  MoveL 2095 to (-402.87, 337.02, -18.74) mm, rotated rx -180 ry 0 rz 0.01 deg; joints [35.505, -31.649, 74.768, -134.161, 54.079, 149.801]
  MoveL 2096 to (-403.75, 334.43, -18.84) mm, rotated rx -180 ry 0 rz 0.01 deg; joints [35.421, -31.691, 74.866, -134.279, 54.073, 149.904]
  MoveL 2097 to (-403.78, 333.95, -18.85) mm, rotated rx -180 ry 0 rz 0.01 deg; joints [35.407, -31.706, 74.899, -134.302, 54.079, 149.928]
  MoveL 2098 to (-403.79, 333.65, -18.86) mm, rotated rx -180 ry 0 rz 0.01 deg; joints [35.399, -31.715, 74.92, -134.317, 54.083, 149.943]
  MoveL 2099 to (-403.79, 333.05, -18.88) mm, rotated rx -180 ry 0 rz 0.01 deg; joints [35.384, -31.736, 74.964, -134.346, 54.091, 149.974]
  MoveL 2100 to (-401.25, 328.08, -19.09) mm, rotated rx 180 ry 0 rz 0.01 deg; joints [35.3, -32.028, 75.587, -134.605, 54.28, 150.319]
  MoveL 2101 to (-395.74, 327.2, -19.29) mm, rotated rx -180 ry 0 rz 0.01 deg; joints [35.38, -32.323, 76.213, -134.688, 54.554, 150.557]
  MoveL 2102 to (-391.79, 331.15, -19.49) mm, rotated rx 180 ry 0 rz 0.01 deg; joints [35.56, -32.373, 76.328, -134.532, 54.691, 150.502]
  MoveL 2103 to (-392.66, 336.66, -19.69) mm, rotated rx -180 ry 0 rz 0.01 deg; joints [35.689, -32.13, 75.838, -134.27, 54.584, 150.205]
  MoveL 2104 to (-397.64, 339.2, -19.9) mm, rotated rx 180 ry 0 rz 0.01 deg; joints [35.662, -31.785, 75.142, -134.119, 54.326, 149.913]
  MoveL 2105 to (-398.51, 339.2, -19.93) mm, rotated rx -180 ry 0 rz 0.01 deg; joints [35.645, -31.741, 75.052, -134.113, 54.286, 149.884]
  MoveL 2106 to (-399.34, 339.13, -19.95) mm, rotated rx 180 ry 0 rz 0.01 deg; joints [35.628, -31.7, 74.972, -134.111, 54.249, 149.859]
  MoveL 2107 to (-399.69, 339.08, -19.97) mm, rotated rx 180 ry 0 rz 0.01 deg; joints [35.62, -31.684, 74.939, -134.111, 54.233, 149.85]
  MoveL 2108 to (-400.55, 338.85, -20) mm, rotated rx 180 ry 0 rz 0.01 deg; joints [35.598, -31.647, 74.867, -134.116, 54.197, 149.832]
  MoveL 2109 to (-400.6, 338.83, -20) mm, rotated rx 180 ry 0 rz 0.01 deg; joints [35.596, -31.646, 74.864, -134.116, 54.195, 149.832]
  MoveL 2110 to (-400.13, 339.01, -20) mm, rotated rx 180 ry 0 rz 0.01 deg; joints [35.61, -31.663, 74.899, -134.112, 54.215, 149.839]
  MoveL 2111 to (-398.92, 339.2, -20) mm, rotated rx 180 ry 0 rz 0.01 deg; joints [35.637, -31.717, 75.009, -134.112, 54.269, 149.872]
  MoveL 2112 to (-213.2, 339.2, -20) mm, rotated rx 180 ry 0 rz 0.01 deg; joints [39.463, -39.848, 91.814, -134.031, 62.159, 155.085]
  MoveL 2113 to (-213.59, 339.14, -20) mm, rotated rx 180 ry 0 rz 0.01 deg; joints [39.452, -39.834, 91.787, -134.036, 62.144, 155.079]
  MoveL 2114 to (-214.1, 339.03, -20) mm, rotated rx 180 ry 0 rz 0.01 deg; joints [39.438, -39.818, 91.754, -134.044, 62.126, 155.072]
  MoveL 2115 to (-215.18, 338.68, -20) mm, rotated rx 180 ry 0 rz 0.01 deg; joints [39.404, -39.787, 91.689, -134.066, 62.088, 155.061]
  MoveL 2116 to (-215.68, 338.49, -20) mm, rotated rx -180 ry 0 rz 0.01 deg; joints [39.388, -39.774, 91.662, -134.077, 62.071, 155.058]
  MoveL 2117 to (-226.92, 332.89, -20) mm, rotated rx 180 ry 0 rz 0.01 deg; joints [38.984, -39.51, 91.121, -134.381, 61.699, 155.03]
  MoveL 2118 to (-227.59, 332.45, -20) mm, rotated rx -180 ry 0 rz 0.01 deg; joints [38.958, -39.497, 91.095, -134.403, 61.678, 155.033]
  MoveL 2119 to (-228.68, 331.54, -20) mm, rotated rx 180 ry 0 rz 0.01 deg; joints [38.909, -39.483, 91.066, -134.448, 61.646, 155.045]
  MoveL 2120 to (-228.85, 331.38, -20) mm, rotated rx 180 ry 0 rz 0.01 deg; joints [38.901, -39.481, 91.062, -134.455, 61.641, 155.048]
  MoveL 2121 to (-237.26, 323.26, -20) mm, rotated rx -180 ry 0 rz 0.01 deg; joints [38.493, -39.4, 90.906, -134.842, 61.408, 155.189]
  MoveL 2122 to (-237.74, 322.68, -20) mm, rotated rx -180 ry 0 rz 0.01 deg; joints [38.467, -39.399, 90.905, -134.869, 61.396, 155.202]
  MoveL 2123 to (-238.69, 321.23, -20) mm, rotated rx -180 ry 0 rz 0.01 deg; joints [38.406, -39.406, 90.921, -134.934, 61.376, 155.24]
  MoveL 2124 to (-238.83, 321, -20) mm, rotated rx -180 ry 0 rz 0.01 deg; joints [38.397, -39.407, 90.925, -134.945, 61.373, 155.247]
  MoveL 2125 to (-243.98, 311.57, -20) mm, rotated rx 180 ry 0 rz 0.01 deg; joints [38.024, -39.491, 91.112, -135.366, 61.284, 155.517]
  MoveL 2126 to (-244.14, 311.23, -20) mm, rotated rx -180 ry 0 rz 0.01 deg; joints [38.011, -39.495, 91.121, -135.381, 61.281, 155.527]
  MoveL 2127 to (-244.73, 309.78, -20) mm, rotated rx 180 ry 0 rz 0.01 deg; joints [37.958, -39.515, 91.165, -135.445, 61.275, 155.573]
  MoveL 2128 to (-244.95, 309.01, -20) mm, rotated rx 180 ry 0 rz 0.01 deg; joints [37.932, -39.53, 91.197, -135.478, 61.276, 155.6]
  MoveL 2129 to (-246.39, 299.58, -20) mm, rotated rx 180 ry 0 rz 0.01 deg; joints [37.638, -39.756, 91.681, -135.879, 61.334, 155.954]
  MoveL 2130 to (-246.42, 299.36, -20) mm, rotated rx 180 ry 0 rz 0.01 deg; joints [37.631, -39.761, 91.692, -135.888, 61.335, 155.962]
  MoveL 2131 to (-246.51, 298.27, -20) mm, rotated rx -180 ry 0 rz 0.01 deg; joints [37.599, -39.79, 91.754, -135.934, 61.345, 156.004]
  MoveC 2132 to (-246.51, 297.75, -20) mm, rotated rx -180 ry 0 rz 0.01 deg; joints [37.584, -39.805, 91.786, -135.956, 61.351, 156.025] to (-246.44, 297.23, -20) mm, rotated rx -180 ry 0 rz 0.01 deg; joints [37.572, -39.824, 91.825, -135.977, 61.36, 156.048]
  MoveL 2133 to (-245.04, 291.02, -20) mm, rotated rx 180 ry 0 rz 0.01 deg; joints [37.427, -40.063, 92.332, -136.227, 61.492, 156.332]
  MoveL 2134 to (-245.03, 290.96, -20) mm, rotated rx 180 ry 0 rz 0.01 deg; joints [37.426, -40.065, 92.337, -136.229, 61.493, 156.335]
  MoveL 2135 to (-244.07, 287.02, -20) mm, rotated rx 180 ry 0 rz 0.01 deg; joints [37.336, -40.219, 92.663, -136.387, 61.579, 156.515]
  MoveL 2136 to (-243.75, 286.2, -20) mm, rotated rx -180 ry 0 rz 0.01 deg; joints [37.319, -40.255, 92.74, -136.418, 61.602, 156.555]
  MoveL 2137 to (-242.37, 283.67, -20) mm, rotated rx 180 ry 0 rz 0.01 deg; joints [37.277, -40.384, 93.011, -136.515, 61.688, 156.688]
  MoveL 2138 to (-242.16, 283.33, -20) mm, rotated rx -180 ry 0 rz 0.01 deg; joints [37.272, -40.402, 93.049, -136.527, 61.7, 156.706]
  MoveL 2139 to (-239.17, 279.09, -20) mm, rotated rx -180 ry 0 rz 0.01 deg; joints [37.217, -40.642, 93.556, -136.683, 61.871, 156.942]
  MoveL 2140 to (-239, 278.88, -20) mm, rotated rx -180 ry 0 rz 0.01 deg; joints [37.214, -40.655, 93.583, -136.691, 61.88, 156.954]
  MoveL 2141 to (-237.09, 276.58, -20) mm, rotated rx -180 ry 0 rz 0.01 deg; joints [37.19, -40.796, 93.879, -136.773, 61.983, 157.087]
  MoveL 2142 to (-236.75, 276.23, -20) mm, rotated rx -180 ry 0 rz 0.01 deg; joints [37.187, -40.819, 93.928, -136.785, 62.001, 157.108]
  MoveL 2143 to (-236.39, 275.91, -20) mm, rotated rx -180 ry 0 rz 0.01 deg; joints [37.186, -40.842, 93.978, -136.796, 62.02, 157.129]
  MoveL 2144 to (-236.08, 275.67, -20) mm, rotated rx 180 ry 0 rz 0.01 deg; joints [37.186, -40.861, 94.018, -136.804, 62.034, 157.146]
  MoveL 2145 to (-232.45, 273.09, -20) mm, rotated rx -180 ry 0 rz 0.01 deg; joints [37.191, -41.076, 94.469, -136.884, 62.209, 157.326]
  MoveL 2146 to (-232.33, 273.01, -20) mm, rotated rx -180 ry 0 rz 0.01 deg; joints [37.191, -41.083, 94.484, -136.886, 62.215, 157.332]
  MoveL 2147 to (-229.06, 270.9, -20) mm, rotated rx -180 ry 0 rz 0.01 deg; joints [37.202, -41.269, 94.876, -136.949, 62.37, 157.486]
  MoveL 2148 to (-228.75, 270.72, -20) mm, rotated rx 180 ry 0 rz 0.01 deg; joints [37.203, -41.287, 94.912, -136.954, 62.384, 157.499]
  MoveL 2149 to (-227.17, 269.93, -20) mm, rotated rx -180 ry 0 rz 0.01 deg; joints [37.215, -41.37, 95.087, -136.975, 62.456, 157.564]
  MoveL 2150 to (-226.77, 269.76, -20) mm, rotated rx -180 ry 0 rz 0.01 deg; joints [37.219, -41.39, 95.129, -136.979, 62.474, 157.579]
  MoveL 2151 to (-224.72, 269.04, -20) mm, rotated rx 180 ry 0 rz 0.01 deg; joints [37.243, -41.489, 95.337, -136.993, 62.563, 157.651]
  MoveL 2152 to (-224.25, 268.91, -20) mm, rotated rx 180 ry 0 rz 0.01 deg; joints [37.25, -41.511, 95.383, -136.994, 62.583, 157.667]
  MoveL 2153 to (-219.17, 267.91, -20) mm, rotated rx -180 ry 0 rz 0.01 deg; joints [37.332, -41.733, 95.848, -136.995, 62.794, 157.813]
  MoveL 2154 to (-218.97, 267.88, -20) mm, rotated rx 180 ry 0 rz 0.01 deg; joints [37.336, -41.742, 95.866, -136.994, 62.802, 157.819]
  MoveL 2155 to (-215.35, 267.39, -20) mm, rotated rx 180 ry 0 rz 0.01 deg; joints [37.401, -41.893, 96.184, -136.985, 62.95, 157.914]
  MoveL 2156 to (-214.9, 267.36, -20) mm, rotated rx 180 ry 0 rz 0.01 deg; joints [37.41, -41.911, 96.221, -136.982, 62.967, 157.925]
  MoveL 2157 to (-178.62, 267.36, -20) mm, rotated rx 180 ry 0 rz 0.01 deg; joints [38.225, -43.259, 99.04, -136.644, 64.36, 158.668]
  MoveL 2158 to (-178.17, 267.39, -20) mm, rotated rx 180 ry 0 rz 0.01 deg; joints [38.236, -43.275, 99.073, -136.639, 64.376, 158.676]
  MoveL 2159 to (-174.54, 267.88, -20) mm, rotated rx 180 ry 0 rz 0.01 deg; joints [38.334, -43.393, 99.32, -136.581, 64.507, 158.73]
  MoveL 2160 to (-174.34, 267.91, -20) mm, rotated rx -180 ry 0 rz 0.01 deg; joints [38.339, -43.399, 99.333, -136.578, 64.515, 158.733]
  MoveL 2161 to (-169.26, 268.91, -20) mm, rotated rx 180 ry 0 rz 0.01 deg; joints [38.485, -43.555, 99.658, -136.484, 64.694, 158.797]
  MoveL 2162 to (-168.86, 269.01, -20) mm, rotated rx 180 ry 0 rz 0.01 deg; joints [38.497, -43.567, 99.683, -136.476, 64.707, 158.801]
  MoveL 2163 to (-167.47, 269.46, -20) mm, rotated rx -180 ry 0 rz 0.01 deg; joints [38.542, -43.604, 99.76, -136.443, 64.754, 158.811]
  MoveL 2164 to (-167.13, 269.6, -20) mm, rotated rx -180 ry 0 rz 0.01 deg; joints [38.554, -43.613, 99.778, -136.434, 64.765, 158.813]
  MoveL 2165 to (-165.28, 270.43, -20) mm, rotated rx -180 ry 0 rz 0.01 deg; joints [38.621, -43.656, 99.867, -136.38, 64.824, 158.818]
  MoveL 2166 to (-164.86, 270.66, -20) mm, rotated rx -180 ry 0 rz 0.01 deg; joints [38.638, -43.665, 99.885, -136.366, 64.837, 158.818]
  MoveL 2167 to (-161.56, 272.76, -20) mm, rotated rx -180 ry 0 rz 0.01 deg; joints [38.775, -43.724, 100.007, -136.246, 64.935, 158.804]
  MoveL 2168 to (-161.46, 272.83, -20) mm, rotated rx -180 ry 0 rz 0.01 deg; joints [38.78, -43.726, 100.01, -136.242, 64.938, 158.803]
  MoveL 2169 to (-158.56, 274.83, -20) mm, rotated rx 180 ry 0 rz 0.01 deg; joints [38.905, -43.774, 100.107, -136.13, 65.022, 158.786]
  MoveL 2170 to (-158.4, 274.95, -20) mm, rotated rx -180 ry 0 rz 0.01 deg; joints [38.913, -43.776, 100.112, -136.124, 65.026, 158.784]
  MoveL 2171 to (-156.94, 276.09, -20) mm, rotated rx -180 ry 0 rz 0.01 deg; joints [38.98, -43.796, 100.153, -136.062, 65.067, 158.77]
  MoveL 2172 to (-156.45, 276.55, -20) mm, rotated rx -180 ry 0 rz 0.01 deg; joints [39.005, -43.801, 100.161, -136.038, 65.079, 158.762]
  MoveL 2173 to (-155.01, 278.23, -20) mm, rotated rx 180 ry 0 rz 0.01 deg; joints [39.087, -43.805, 100.167, -135.954, 65.112, 158.728]
  MoveL 2174 to (-154.82, 278.47, -20) mm, rotated rx 180 ry 0 rz 0.01 deg; joints [39.098, -43.805, 100.166, -135.943, 65.116, 158.722]
  MoveL 2175 to (-151.36, 283.31, -20) mm, rotated rx 180 ry 0 rz 0.01 deg; joints [39.32, -43.791, 100.13, -135.711, 65.185, 158.608]
  MoveL 2176 to (-151.14, 283.67, -20) mm, rotated rx 180 ry 0 rz 0.01 deg; joints [39.335, -43.789, 100.125, -135.694, 65.189, 158.599]
  MoveL 2177 to (-149.76, 286.2, -20) mm, rotated rx 180 ry 0 rz 0.01 deg; joints [39.441, -43.766, 100.073, -135.577, 65.209, 158.531]
  MoveL 2178 to (-149.44, 287.04, -20) mm, rotated rx -180 ry 0 rz 0.01 deg; joints [39.472, -43.753, 100.045, -135.541, 65.211, 158.505]
  MoveL 2179 to (-147.12, 296.83, -20) mm, rotated rx -180 ry 0 rz 0.01 deg; joints [39.807, -43.556, 99.616, -135.125, 65.177, 158.18]
  MoveL 2180 to (-147.03, 297.45, -20) mm, rotated rx 180 ry 0 rz 0.01 deg; joints [39.827, -43.541, 99.584, -135.1, 65.173, 158.158]
  MoveL 2181 to (-146.99, 298.18, -20) mm, rotated rx 180 ry 0 rz 0.01 deg; joints [39.849, -43.521, 99.542, -135.071, 65.165, 158.131]
  MoveL 2182 to (-147.03, 298.84, -20) mm, rotated rx 180 ry 0 rz 0.01 deg; joints [39.867, -43.501, 99.498, -135.045, 65.156, 158.105]
  MoveL 2183 to (-148.48, 308.63, -20) mm, rotated rx 180 ry 0 rz 0.01 deg; joints [40.11, -43.165, 98.78, -134.673, 64.983, 157.7]
  MoveL 2184 to (-148.62, 309.22, -20) mm, rotated rx 180 ry 0 rz 0.01 deg; joints [40.123, -43.143, 98.732, -134.651, 64.971, 157.674]
  MoveL 2185 to (-149.12, 310.67, -20) mm, rotated rx 180 ry 0 rz 0.01 deg; joints [40.152, -43.083, 98.605, -134.599, 64.935, 157.608]
  MoveL 2186 to (-149.35, 311.2, -20) mm, rotated rx -180 ry 0 rz 0.01 deg; joints [40.161, -43.059, 98.554, -134.581, 64.92, 157.583]
  MoveL 2187 to (-154.68, 321, -20) mm, rotated rx -180 ry 0 rz 0.01 deg; joints [40.31, -42.579, 97.535, -134.25, 64.603, 157.092]
  MoveL 2188 to (-154.82, 321.23, -20) mm, rotated rx -180 ry 0 rz 0.01 deg; joints [40.313, -42.567, 97.51, -134.242, 64.595, 157.08]
  MoveL 2189 to (-155.77, 322.68, -20) mm, rotated rx 180 ry 0 rz 0.01 deg; joints [40.331, -42.49, 97.346, -134.195, 64.542, 157.003]
  MoveL 2190 to (-156.25, 323.26, -20) mm, rotated rx 180 ry 0 rz 0.01 deg; joints [40.336, -42.455, 97.274, -134.177, 64.518, 156.971]
  MoveL 2191 to (-163.72, 330.51, -20) mm, rotated rx 180 ry 0 rz 0.01 deg; joints [40.361, -41.967, 96.243, -133.964, 64.151, 156.527]
  MoveL 2192 to (-163.84, 330.62, -20) mm, rotated rx 180 ry 0 rz 0.01 deg; joints [40.361, -41.96, 96.227, -133.961, 64.145, 156.521]
  MoveL 2193 to (-165.86, 332.4, -20) mm, rotated rx -180 ry 0 rz 0.01 deg; joints [40.363, -41.832, 95.959, -133.91, 64.048, 156.407]
  MoveL 2194 to (-166.59, 332.89, -20) mm, rotated rx 180 ry 0 rz 0.01 deg; joints [40.359, -41.791, 95.872, -133.897, 64.015, 156.372]
  MoveL 2195 to (-177.84, 338.49, -20) mm, rotated rx 180 ry 0 rz 0.01 deg; joints [40.25, -41.207, 94.645, -133.779, 63.524, 155.905]
  MoveL 2196 to (-178.19, 338.64, -20) mm, rotated rx -180 ry 0 rz 0.01 deg; joints [40.246, -41.189, 94.608, -133.776, 63.508, 155.891]
  MoveL 2197 to (-178.92, 338.9, -20) mm, rotated rx -180 ry 0 rz 0.01 deg; joints [40.237, -41.154, 94.535, -133.772, 63.478, 155.865]
  MoveL 2198 to (-179.55, 339.06, -20) mm, rotated rx 180 ry 0 rz 0.01 deg; joints [40.227, -41.126, 94.475, -133.771, 63.452, 155.844]
  MoveL 2199 to (-180.47, 339.2, -20) mm, rotated rx -180 ry 0 rz 0.01 deg; joints [40.209, -41.087, 94.395, -133.773, 63.415, 155.818]
  MoveL 2200 to (4.87, 339.21, -20) mm, rotated rx -180 ry 0 rz 0.01 deg; joints [44.909, -47.308, 107.456, -131.259, 69.938, 159.405]
  MoveL 2201 to (5.94, 339.15, -20) mm, rotated rx 180 ry 0 rz 0.01 deg; joints [44.937, -47.342, 107.529, -131.242, 69.974, 159.426]
  MoveL 2202 to (6.8, 338.95, -20) mm, rotated rx 180 ry 0 rz 0.01 deg; joints [44.955, -47.374, 107.597, -131.233, 70.004, 159.448]
  MoveL 2203 to (7.07, 338.84, -20) mm, rotated rx 180 ry 0 rz 0.01 deg; joints [44.96, -47.386, 107.621, -131.233, 70.014, 159.457]
  MoveL 2204 to (7.37, 338.63, -20) mm, rotated rx 180 ry 0 rz 0.01 deg; joints [44.962, -47.401, 107.654, -131.235, 70.027, 159.47]
  MoveL 2205 to (9.66, 336.38, -20) mm, rotated rx -180 ry 0 rz 0.01 deg; joints [44.963, -47.537, 107.944, -131.276, 70.129, 159.593]
  MoveL 2206 to (9.9, 336.02, -20) mm, rotated rx -180 ry 0 rz 0.01 deg; joints [44.96, -47.554, 107.982, -131.285, 70.141, 159.611]
  MoveL 2207 to (10.07, 335.56, -20) mm, rotated rx -180 ry 0 rz 0.01 deg; joints [44.952, -47.573, 108.023, -131.299, 70.153, 159.631]
  MoveL 2208 to (10.27, 334.35, -20) mm, rotated rx 180 ry 0 rz 0.01 deg; joints [44.923, -47.614, 108.112, -131.34, 70.174, 159.679]
  MoveL 2209 to (10.27, 31.66, -20) mm, rotated rx -180 ry 0 rz 0.01 deg; joints [35.113, -55.058, 124.722, -143.253, 74.093, 169.379]
  MoveL 2210 to (8.9, 37.18, -20) mm, rotated rx 180 ry 0 rz 0.01 deg; joints [35.282, -54.906, 124.374, -143.048, 73.972, 169.208]
  MoveL 2211 to (8.66, 37.84, -20) mm, rotated rx 180 ry 0 rz 0.01 deg; joints [35.3, -54.885, 124.327, -143.024, 73.955, 169.186]
  MoveL 2212 to (8, 39.21, -20) mm, rotated rx -180 ry 0 rz 0.01 deg; joints [35.334, -54.837, 124.219, -142.98, 73.913, 169.138]
  MoveL 2213 to (7.84, 39.5, -20) mm, rotated rx -180 ry 0 rz 0.01 deg; joints [35.34, -54.827, 124.195, -142.971, 73.904, 169.128]
  MoveL 2214 to (2.04, 49.03, -20) mm, rotated rx -180 ry 0 rz 0.01 deg; joints [35.539, -54.458, 123.362, -142.687, 73.577, 168.778]
  MoveL 2215 to (1.81, 49.36, -20) mm, rotated rx -180 ry 0 rz 0.01 deg; joints [35.545, -54.444, 123.332, -142.678, 73.565, 168.765]
  MoveL 2216 to (0.94, 50.47, -20) mm, rotated rx -180 ry 0 rz 0.01 deg; joints [35.563, -54.395, 123.221, -142.649, 73.52, 168.721]
  MoveL 2217 to (0.39, 51.02, -20) mm, rotated rx -180 ry 0 rz 0.01 deg; joints [35.569, -54.367, 123.159, -142.637, 73.494, 168.697]
  MoveL 2218 to (-7.44, 57.3, -20) mm, rotated rx -180 ry 0 rz 0.01 deg; joints [35.593, -54, 122.339, -142.53, 73.141, 168.403]
  MoveL 2219 to (-7.81, 57.56, -20) mm, rotated rx 180 ry 0 rz 0.01 deg; joints [35.593, -53.983, 122.302, -142.526, 73.125, 168.39]
  MoveL 2220 to (-8.48, 57.96, -20) mm, rotated rx 180 ry 0 rz 0.01 deg; joints [35.59, -53.954, 122.239, -142.523, 73.096, 168.369]
  MoveL 2221 to (-9.25, 58.3, -20) mm, rotated rx 180 ry 0 rz 0.01 deg; joints [35.583, -53.924, 122.171, -142.523, 73.065, 168.348]
  MoveL 2222 to (-19.1, 61.27, -20) mm, rotated rx -180 ry 0 rz 0.01 deg; joints [35.436, -53.56, 121.37, -142.591, 72.685, 168.115]
  MoveL 2223 to (-19.98, 61.41, -20) mm, rotated rx -180 ry 0 rz 0.01 deg; joints [35.419, -53.53, 121.304, -142.601, 72.652, 168.098]
  MoveL 2224 to (-22.52, 61.49, -20) mm, rotated rx 180 ry 0 rz 0.01 deg; joints [35.357, -53.45, 121.13, -142.647, 72.563, 168.057]
  MoveL 2225 to (-22.91, 61.48, -20) mm, rotated rx 180 ry 0 rz 0.01 deg; joints [35.346, -53.438, 121.104, -142.655, 72.549, 168.051]
  MoveL 2226 to (-28.72, 60.97, -20) mm, rotated rx 180 ry 0 rz 0.01 deg; joints [35.181, -53.269, 120.736, -142.785, 72.353, 167.978]
  MoveL 2227 to (-29.06, 60.92, -20) mm, rotated rx -180 ry 0 rz 0.01 deg; joints [35.171, -53.259, 120.715, -142.794, 72.342, 167.974]
  MoveL 2228 to (-31.97, 60.36, -20) mm, rotated rx -180 ry 0 rz 0.01 deg; joints [35.077, -53.181, 120.545, -142.872, 72.247, 167.946]
  MoveL 2229 to (-32.71, 60.13, -20) mm, rotated rx 180 ry 0 rz 0.01 deg; joints [35.05, -53.163, 120.506, -142.895, 72.224, 167.942]
  MoveL 2230 to (-36.58, 58.38, -20) mm, rotated rx 180 ry 0 rz 0.01 deg; joints [34.891, -53.078, 120.325, -143.04, 72.11, 167.933]
  MoveL 2231 to (-36.74, 58.31, -20) mm, rotated rx 180 ry 0 rz 0.01 deg; joints [34.884, -53.075, 120.318, -143.046, 72.106, 167.932]
  MoveL 2232 to (-40.59, 56.33, -20) mm, rotated rx 180 ry 0 rz 0.01 deg; joints [34.717, -52.995, 120.149, -143.199, 71.996, 167.93]
  MoveL 2233 to (-40.91, 56.15, -20) mm, rotated rx -180 ry 0 rz 0.01 deg; joints [34.703, -52.989, 120.136, -143.212, 71.987, 167.931]
  MoveL 2234 to (-42.32, 55.22, -20) mm, rotated rx 180 ry 0 rz 0.01 deg; joints [34.635, -52.964, 120.084, -143.276, 71.949, 167.936]
  MoveL 2235 to (-42.64, 54.98, -20) mm, rotated rx -180 ry 0 rz 0.01 deg; joints [34.618, -52.959, 120.073, -143.292, 71.941, 167.938]
  MoveL 2236 to (-44.19, 53.67, -20) mm, rotated rx 180 ry 0 rz 0.01 deg; joints [34.533, -52.937, 120.029, -143.376, 71.903, 167.952]
  MoveL 2237 to (-44.56, 53.31, -20) mm, rotated rx -180 ry 0 rz 0.01 deg; joints [34.511, -52.933, 120.021, -143.397, 71.894, 167.956]
  MoveL 2238 to (-48.48, 48.82, -20) mm, rotated rx -180 ry 0 rz 0.01 deg; joints [34.253, -52.901, 119.962, -143.656, 71.812, 168.024]
  MoveL 2239 to (-48.63, 48.64, -20) mm, rotated rx 180 ry 0 rz 0.01 deg; joints [34.243, -52.9, 119.96, -143.666, 71.81, 168.027]
  MoveL 2240 to (-50.41, 46.31, -20) mm, rotated rx 180 ry 0 rz 0.01 deg; joints [34.115, -52.892, 119.947, -143.796, 71.776, 168.066]
  MoveL 2241 to (-50.64, 45.95, -20) mm, rotated rx 180 ry 0 rz 0.01 deg; joints [34.097, -52.892, 119.947, -143.815, 71.772, 168.073]
  MoveL 2242 to (-68.79, 14.55, -20) mm, rotated rx 180 ry 0 rz 0.01 deg; joints [32.519, -52.939, 120.118, -145.458, 71.518, 168.675]
  MoveL 2243 to (-69, 14.13, -20) mm, rotated rx -180 ry 0 rz 0.01 deg; joints [32.499, -52.94, 120.122, -145.479, 71.516, 168.684]
  MoveL 2244 to (-70.62, 10.14, -20) mm, rotated rx -180 ry 0 rz 0.01 deg; joints [32.314, -52.965, 120.185, -145.677, 71.507, 168.769]
  MoveL 2245 to (-70.69, 9.97, -20) mm, rotated rx -180 ry 0 rz 0.01 deg; joints [32.306, -52.966, 120.189, -145.685, 71.507, 168.773]
  MoveL 2246 to (-72.18, 5.61, -20) mm, rotated rx 180 ry 0 rz 0.01 deg; joints [32.11, -53.002, 120.276, -145.896, 71.507, 168.869]
  MoveL 2247 to (-72.29, 5.22, -20) mm, rotated rx -180 ry 0 rz 0.01 deg; joints [32.093, -53.006, 120.285, -145.915, 71.508, 168.878]
  MoveL 2248 to (-72.6, 3.77, -20) mm, rotated rx -180 ry 0 rz 0.01 deg; joints [32.033, -53.024, 120.327, -145.982, 71.515, 168.913]
  MoveL 2249 to (-72.66, 3.4, -20) mm, rotated rx -180 ry 0 rz 0.01 deg; joints [32.017, -53.029, 120.34, -145.999, 71.518, 168.923]
  MoveL 2250 to (-72.87, 1.22, -20) mm, rotated rx 180 ry 0 rz 0.01 deg; joints [31.932, -53.064, 120.42, -146.096, 71.537, 168.978]
  MoveL 2251 to (-72.89, 0.7, -20) mm, rotated rx -180 ry 0 rz 0.01 deg; joints [31.912, -53.073, 120.442, -146.118, 71.543, 168.992]
  MoveL 2252 to (-72.52, -5.83, -20) mm, rotated rx -180 ry 0 rz 0.01 deg; joints [31.677, -53.209, 120.753, -146.392, 71.639, 169.173]
  MoveL 2253 to (-72.5, -6.03, -20) mm, rotated rx -180 ry 0 rz 0.01 deg; joints [31.67, -53.213, 120.762, -146.4, 71.642, 169.179]
  MoveL 2254 to (-72.25, -8.21, -20) mm, rotated rx -180 ry 0 rz 0.01 deg; joints [31.595, -53.262, 120.874, -146.49, 71.679, 169.241]
  MoveL 2255 to (-72.16, -8.69, -20) mm, rotated rx 180 ry 0 rz 0.01 deg; joints [31.579, -53.274, 120.901, -146.509, 71.688, 169.255]
  MoveL 2256 to (-71.97, -9.41, -20) mm, rotated rx 180 ry 0 rz 0.01 deg; joints [31.556, -53.294, 120.946, -146.537, 71.704, 169.277]
  MoveL 2257 to (-71.86, -9.75, -20) mm, rotated rx 180 ry 0 rz 0.01 deg; joints [31.546, -53.304, 120.969, -146.55, 71.712, 169.288]
  MoveL 2258 to (-70.76, -12.61, -20) mm, rotated rx 180 ry 0 rz 0.01 deg; joints [31.464, -53.393, 121.169, -146.654, 71.788, 169.38]
  MoveL 2259 to (-70.67, -12.82, -20) mm, rotated rx 180 ry 0 rz 0.01 deg; joints [31.458, -53.399, 121.184, -146.662, 71.794, 169.387]
  MoveL 2260 to (-68.64, -17.22, -20) mm, rotated rx 180 ry 0 rz 0.01 deg; joints [31.339, -53.546, 121.516, -146.817, 71.924, 169.532]
  MoveL 2261 to (-68.49, -17.51, -20) mm, rotated rx -180 ry 0 rz 0.01 deg; joints [31.332, -53.557, 121.539, -146.827, 71.933, 169.542]
  MoveL 2262 to (-67.65, -18.96, -20) mm, rotated rx -180 ry 0 rz 0.01 deg; joints [31.297, -53.611, 121.66, -146.876, 71.982, 169.593]
  MoveL 2263 to (-67.51, -19.16, -20) mm, rotated rx -180 ry 0 rz 0.01 deg; joints [31.292, -53.619, 121.678, -146.882, 71.99, 169.6]
  MoveL 2264 to (-66.75, -20.28, -20) mm, rotated rx -180 ry 0 rz 0.01 deg; joints [31.267, -53.664, 121.78, -146.918, 72.032, 169.64]
  MoveL 2265 to (-66.28, -20.83, -20) mm, rotated rx 180 ry 0 rz 0.01 deg; joints [31.257, -53.689, 121.836, -146.933, 72.056, 169.662]
  MoveL 2266 to (-59.77, -26.97, -20) mm, rotated rx -180 ry 0 rz 0.01 deg; joints [31.174, -54.01, 122.554, -147.089, 72.372, 169.916]
  MoveL 2267 to (-59.61, -27.11, -20) mm, rotated rx -180 ry 0 rz 0.01 deg; joints [31.172, -54.018, 122.571, -147.092, 72.379, 169.922]
  MoveL 2268 to (-58.52, -28.02, -20) mm, rotated rx 180 ry 0 rz 0.01 deg; joints [31.163, -54.069, 122.685, -147.112, 72.431, 169.961]
  MoveC 2269 to (-58.09, -28.32, -20) mm, rotated rx -180 ry 0 rz 0.01 deg; joints [31.161, -54.088, 122.729, -147.118, 72.45, 169.975] to (-57.61, -28.56, -20) mm, rotated rx 180 ry 0 rz 0.01 deg; joints [31.163, -54.108, 122.772, -147.12, 72.471, 169.988]
  MoveL 2270 to (-50.81, -31.27, -20) mm, rotated rx 180 ry 0 rz 0.01 deg; joints [31.217, -54.373, 123.361, -147.12, 72.753, 170.155]
  MoveL 2271 to (-342.73, -31.27, -20) mm, rotated rx -180 ry 0 rz 0.01 deg; joints [25.548, -43.852, 100.808, -150.481, 61.131, 165.794]
  MoveL 2272 to (-336.29, -28.75, -20) mm, rotated rx -180 ry 0 rz 0.01 deg; joints [25.738, -44.068, 101.258, -150.336, 61.385, 165.824]
  MoveL 2273 to (-335.78, -28.51, -20) mm, rotated rx -180 ry 0 rz 0.01 deg; joints [25.754, -44.084, 101.292, -150.323, 61.405, 165.825]
  MoveL 2274 to (-335.06, -28.07, -20) mm, rotated rx 180 ry 0 rz 0.01 deg; joints [25.781, -44.106, 101.336, -150.3, 61.432, 165.823]
  MoveL 2275 to (-334.48, -27.64, -20) mm, rotated rx 180 ry 0 rz 0.01 deg; joints [25.805, -44.121, 101.367, -150.278, 61.452, 165.82]
  MoveL 2276 to (-329.12, -22.62, -20) mm, rotated rx 180 ry 0 rz 0.01 deg; joints [26.062, -44.244, 101.617, -150.03, 61.631, 165.754]
  MoveL 2277 to (-329.06, -22.56, -20) mm, rotated rx 180 ry 0 rz 0.01 deg; joints [26.066, -44.246, 101.62, -150.027, 61.633, 165.753]
  MoveL 2278 to (-326.88, -20.42, -20) mm, rotated rx 180 ry 0 rz 0.01 deg; joints [26.174, -44.293, 101.716, -149.921, 61.704, 165.723]
  MoveL 2279 to (-326.36, -19.74, -20) mm, rotated rx 180 ry 0 rz 0.01 deg; joints [26.206, -44.302, 101.733, -149.889, 61.72, 165.711]
  MoveL 2280 to (-325.04, -17.54, -20) mm, rotated rx 180 ry 0 rz 0.01 deg; joints [26.302, -44.313, 101.753, -149.786, 61.753, 165.665]
  MoveL 2281 to (-324.87, -17.22, -20) mm, rotated rx 180 ry 0 rz 0.01 deg; joints [26.316, -44.314, 101.754, -149.771, 61.757, 165.658]
  MoveL 2282 to (-322.51, -12.1, -20) mm, rotated rx 180 ry 0 rz 0.01 deg; joints [26.527, -44.312, 101.738, -149.536, 61.804, 165.539]
  MoveL 2283 to (-322.39, -11.81, -20) mm, rotated rx -180 ry 0 rz 0.01 deg; joints [26.539, -44.311, 101.736, -149.523, 61.806, 165.532]
  MoveL 2284 to (-321.51, -9.31, -20) mm, rotated rx -180 ry 0 rz 0.01 deg; joints [26.639, -44.298, 101.705, -149.409, 61.817, 165.469]
  MoveL 2285 to (-321.34, -8.61, -20) mm, rotated rx -180 ry 0 rz 0.01 deg; joints [26.665, -44.291, 101.689, -149.379, 61.816, 165.45]
  MoveL 2286 to (-321.02, -6.07, -20) mm, rotated rx -180 ry 0 rz 0.01 deg; joints [26.755, -44.255, 101.609, -149.267, 61.803, 165.377]
  MoveL 2287 to (-321, -5.83, -20) mm, rotated rx 180 ry 0 rz 0.01 deg; joints [26.764, -44.252, 101.6, -149.257, 61.801, 165.369]
  MoveL 2288 to (-320.63, 0.7, -20) mm, rotated rx -180 ry 0 rz 0.01 deg; joints [26.989, -44.139, 101.351, -148.974, 61.747, 165.171]
  MoveL 2289 to (-320.63, 1.14, -20) mm, rotated rx 180 ry 0 rz 0.01 deg; joints [27.004, -44.13, 101.332, -148.955, 61.742, 165.157]
  MoveL 2290 to (-320.74, 2.59, -20) mm, rotated rx 180 ry 0 rz 0.01 deg; joints [27.05, -44.098, 101.26, -148.893, 61.721, 165.11]
  MoveL 2291 to (-320.79, 2.97, -20) mm, rotated rx 180 ry 0 rz 0.01 deg; joints [27.062, -44.088, 101.239, -148.877, 61.715, 165.097]
  MoveL 2292 to (-321.21, 5.15, -20) mm, rotated rx 180 ry 0 rz 0.01 deg; joints [27.128, -44.028, 101.109, -148.786, 61.673, 165.021]
  MoveL 2293 to (-321.33, 5.61, -20) mm, rotated rx -180 ry 0 rz 0.01 deg; joints [27.141, -44.014, 101.079, -148.767, 61.663, 165.004]
  MoveL 2294 to (-322.71, 9.63, -20) mm, rotated rx -180 ry 0 rz 0.01 deg; joints [27.251, -43.879, 100.786, -148.603, 61.56, 164.853]
  MoveL 2295 to (-322.76, 9.77, -20) mm, rotated rx -180 ry 0 rz 0.01 deg; joints [27.255, -43.874, 100.776, -148.597, 61.556, 164.848]
  MoveL 2296 to (-324.33, 13.74, -20) mm, rotated rx 180 ry 0 rz 0.01 deg; joints [27.36, -43.731, 100.468, -148.436, 61.446, 164.694]
  MoveL 2297 to (-324.54, 14.18, -20) mm, rotated rx 180 ry 0 rz 0.01 deg; joints [27.371, -43.714, 100.43, -148.418, 61.432, 164.676]
  MoveL 2298 to (-342.68, 45.66, -20) mm, rotated rx -180 ry 0 rz 0.01 deg; joints [28.088, -42.32, 97.447, -147.162, 60.301, 163.317]
  MoveL 2299 to (-342.91, 46, -20) mm, rotated rx -180 ry 0 rz 0.01 deg; joints [28.095, -42.303, 97.412, -147.148, 60.288, 163.302]
  MoveL 2300 to (-344.86, 48.62, -20) mm, rotated rx -180 ry 0 rz 0.01 deg; joints [28.146, -42.166, 97.12, -147.045, 60.174, 163.177]
  MoveL 2301 to (-345.02, 48.81, -20) mm, rotated rx -180 ry 0 rz 0.01 deg; joints [28.15, -42.156, 97.098, -147.037, 60.165, 163.168]
  MoveL 2302 to (-348.42, 52.74, -20) mm, rotated rx -180 ry 0 rz 0.01 deg; joints [28.217, -41.929, 96.617, -146.883, 59.973, 162.97]
  MoveL 2303 to (-348.65, 52.98, -20) mm, rotated rx 180 ry 0 rz 0.01 deg; joints [28.221, -41.915, 96.586, -146.874, 59.96, 162.957]
  MoveL 2304 to (-350.21, 54.47, -20) mm, rotated rx -180 ry 0 rz 0.01 deg; joints [28.242, -41.817, 96.379, -146.817, 59.875, 162.876]
  MoveL 2305 to (-350.59, 54.77, -20) mm, rotated rx 180 ry 0 rz 0.01 deg; joints [28.245, -41.795, 96.332, -146.805, 59.855, 162.859]
  MoveL 2306 to (-352.04, 55.8, -20) mm, rotated rx -180 ry 0 rz 0.01 deg; joints [28.253, -41.712, 96.156, -146.767, 59.78, 162.796]
  MoveL 2307 to (-352.42, 56.04, -20) mm, rotated rx -180 ry 0 rz 0.01 deg; joints [28.254, -41.69, 96.111, -146.758, 59.761, 162.78]
  MoveL 2308 to (-356.26, 58.05, -20) mm, rotated rx 180 ry 0 rz 0.01 deg; joints [28.252, -41.485, 95.678, -146.687, 59.57, 162.636]
  MoveL 2309 to (-356.43, 58.13, -20) mm, rotated rx -180 ry 0 rz 0.01 deg; joints [28.252, -41.476, 95.659, -146.684, 59.562, 162.63]
  MoveL 2310 to (-360.78, 60.12, -20) mm, rotated rx 180 ry 0 rz 0.01 deg; joints [28.241, -41.248, 95.18, -146.615, 59.348, 162.476]
  MoveL 2311 to (-361.55, 60.36, -20) mm, rotated rx -180 ry 0 rz 0.01 deg; joints [28.236, -41.211, 95.101, -146.607, 59.311, 162.452]
  MoveL 2312 to (-364.45, 60.92, -20) mm, rotated rx 180 ry 0 rz 0.01 deg; joints [28.204, -41.075, 94.816, -146.593, 59.177, 162.375]
  MoveL 2313 to (-364.78, 60.97, -20) mm, rotated rx -180 ry 0 rz 0.01 deg; joints [28.2, -41.06, 94.784, -146.592, 59.162, 162.367]
  MoveL 2314 to (-370.22, 61.47, -20) mm, rotated rx 180 ry 0 rz 0.01 deg; joints [28.123, -40.816, 94.275, -146.588, 58.915, 162.24]
  MoveL 2315 to (-370.61, 61.48, -20) mm, rotated rx 180 ry 0 rz 0.01 deg; joints [28.117, -40.799, 94.239, -146.589, 58.897, 162.232]
  MoveL 2316 to (-373.51, 61.41, -20) mm, rotated rx -180 ry 0 rz 0.01 deg; joints [28.066, -40.676, 93.982, -146.601, 58.769, 162.175]
  MoveL 2317 to (-374.4, 61.27, -20) mm, rotated rx 180 ry 0 rz 0.01 deg; joints [28.047, -40.641, 93.909, -146.61, 58.731, 162.162]
  MoveL 2318 to (-383.58, 58.54, -20) mm, rotated rx -180 ry 0 rz 0.01 deg; joints [27.807, -40.303, 93.21, -146.753, 58.35, 162.071]
  MoveL 2319 to (-383.91, 58.43, -20) mm, rotated rx 180 ry 0 rz 0.01 deg; joints [27.798, -40.292, 93.187, -146.759, 58.336, 162.068]
  MoveL 2320 to (-384.91, 58.01, -20) mm, rotated rx 180 ry 0 rz 0.01 deg; joints [27.769, -40.257, 93.115, -146.78, 58.296, 162.062]
  MoveL 2321 to (-385.73, 57.53, -20) mm, rotated rx -180 ry 0 rz 0.01 deg; joints [27.74, -40.232, 93.064, -146.803, 58.264, 162.062]
  MoveL 2322 to (-393.9, 51.03, -20) mm, rotated rx -180 ry 0 rz 0.01 deg; joints [27.401, -40.018, 92.628, -147.105, 57.967, 162.123]
  MoveL 2323 to (-394.45, 50.47, -20) mm, rotated rx -180 ry 0 rz 0.01 deg; joints [27.374, -40.006, 92.604, -147.13, 57.948, 162.131]
  MoveL 2324 to (-395.32, 49.36, -20) mm, rotated rx -180 ry 0 rz 0.01 deg; joints [27.325, -39.992, 92.576, -147.181, 57.92, 162.152]
  MoveL 2325 to (-395.55, 49.03, -20) mm, rotated rx -180 ry 0 rz 0.01 deg; joints [27.311, -39.989, 92.571, -147.195, 57.913, 162.159]
  MoveL 2326 to (-401.35, 39.5, -20) mm, rotated rx -180 ry 0 rz 0.01 deg; joints [26.916, -39.94, 92.485, -147.624, 57.753, 162.375]
  MoveL 2327 to (-401.51, 39.21, -20) mm, rotated rx -180 ry 0 rz 0.01 deg; joints [26.904, -39.939, 92.484, -147.636, 57.749, 162.381]
  MoveL 2328 to (-402.18, 37.84, -20) mm, rotated rx 180 ry 0 rz 0.01 deg; joints [26.85, -39.939, 92.487, -147.698, 57.734, 162.416]
  MoveL 2329 to (-402.42, 37.18, -20) mm, rotated rx -180 ry 0 rz 0.01 deg; joints [26.825, -39.943, 92.496, -147.727, 57.73, 162.434]
  MoveL 2330 to (-403.78, 31.68, -20) mm, rotated rx -180 ry 0 rz 0.01 deg; joints [26.63, -40, 92.625, -147.97, 57.728, 162.598]
  MoveL 2331 to (-403.79, 333.8, -20) mm, rotated rx -180 ry 0 rz 0.01 deg; joints [35.404, -31.662, 74.905, -134.332, 54.112, 149.974]
  MoveL 2332 to (-403.73, 334.87, -20) mm, rotated rx -180 ry 0 rz 0.01 deg; joints [35.433, -31.628, 74.832, -134.281, 54.1, 149.922]
  MoveL 2333 to (-403.53, 335.74, -20) mm, rotated rx 180 ry 0 rz 0.01 deg; joints [35.46, -31.607, 74.788, -134.241, 54.098, 149.885]
  MoveL 2334 to (-403.42, 336, -20) mm, rotated rx 180 ry 0 rz 0.01 deg; joints [35.469, -31.603, 74.781, -134.229, 54.1, 149.875]
  MoveL 2335 to (-403.03, 336.5, -19.83) mm, rotated rx 180 ry 0 rz 0.01 deg; joints [35.489, -31.612, 74.784, -134.205, 54.107, 149.858]
  MoveL 2336 to (-402.62, 336.71, -19.37) mm, rotated rx 180 ry 0 rz 0.01 deg; joints [35.502, -31.645, 74.813, -134.189, 54.111, 149.846]
  MoveL 2337 to (-402.46, 336.75, -18.73) mm, rotated rx -180 ry 0 rz 0.01 deg; joints [35.506, -31.679, 74.83, -134.176, 54.101, 149.828]
  Set speed (1000.0 mm/s)
  MoveL 2338 to (-402.46, 336.75, 11) mm, rotated rx 180 ry 0 rz 0.01 deg; joints [35.493, -32.912, 74.899, -133.574, 53.288, 148.796]
  Set speed (1000.0 mm/s)
  MoveL 2339 to (-212.83, 109.42, 11) mm, rotated rx 180 ry 0 rz 0.01 deg; joints [32.6, -47.593, 105.133, -143.048, 63.709, 162.556]
  Set speed (100.0 mm/s)
  MoveL 2340 to (-212.83, 109.42, -8.23) mm, rotated rx -180 ry 0 rz 0.01 deg; joints [32.611, -46.607, 105.1, -143.314, 64.475, 163.186]
  MoveL 2341 to (-212.67, 109.4, -8.85) mm, rotated rx 180 ry 0 rz 0.01 deg; joints [32.614, -46.581, 105.112, -143.321, 64.507, 163.209]
  MoveL 2342 to (-212.22, 109.37, -9.32) mm, rotated rx 180 ry 0 rz 0.01 deg; joints [32.623, -46.575, 105.146, -143.324, 64.543, 163.233]
  MoveL 2343 to (-211.61, 109.38, -9.5) mm, rotated rx -180 ry 0 rz 0.01 deg; joints [32.636, -46.588, 105.193, -143.32, 64.574, 163.249]
  MoveL 2344 to (-206.37, 113.41, -9.74) mm, rotated rx 180 ry 0 rz 0.01 deg; joints [32.876, -46.677, 105.398, -143.1, 64.741, 163.215]
  MoveL 2345 to (-207.96, 119.82, -9.99) mm, rotated rx -180 ry 0 rz 0.01 deg; joints [33.051, -46.457, 104.953, -142.853, 64.616, 162.985]
  MoveL 2346 to (-214.47, 120.93, -10.23) mm, rotated rx 180 ry 0 rz 0.01 deg; joints [32.95, -46.177, 104.39, -142.877, 64.359, 162.842]
  MoveL 2347 to (-218.1, 115.41, -10.48) mm, rotated rx -180 ry 0 rz 0.01 deg; joints [32.697, -46.157, 104.384, -143.147, 64.29, 162.97]
  MoveL 2348 to (-214.5, 109.88, -10.72) mm, rotated rx -180 ry 0 rz 0.01 deg; joints [32.593, -46.406, 104.941, -143.345, 64.504, 163.222]
  MoveL 2349 to (-207.98, 110.96, -10.96) mm, rotated rx 180 ry 0 rz 0.01 deg; joints [32.764, -46.61, 105.392, -143.235, 64.755, 163.307]
  MoveL 2350 to (-206.36, 117.36, -11.21) mm, rotated rx 180 ry 0 rz 0.01 deg; joints [33.005, -46.51, 105.197, -142.955, 64.754, 163.133]
  MoveL 2351 to (-211.58, 121.41, -11.45) mm, rotated rx 180 ry 0 rz 0.01 deg; joints [33.027, -46.21, 104.588, -142.844, 64.514, 162.916]
  MoveL 2352 to (-217.38, 118.26, -11.7) mm, rotated rx -180 ry 0 rz 0.01 deg; joints [32.804, -46.055, 104.294, -143.038, 64.333, 162.927]
  MoveL 2353 to (-216.81, 111.68, -11.94) mm, rotated rx -180 ry 0 rz 0.01 deg; joints [32.604, -46.215, 104.667, -143.31, 64.44, 163.162]
  MoveL 2354 to (-210.55, 109.56, -12.18) mm, rotated rx -180 ry 0 rz 0.01 deg; joints [32.665, -46.484, 105.259, -143.337, 64.719, 163.348]
  MoveL 2355 to (-206.11, 114.44, -12.43) mm, rotated rx 180 ry 0 rz 0.01 deg; joints [32.917, -46.523, 105.359, -143.09, 64.845, 163.272]
  MoveL 2356 to (-208.8, 120.47, -12.67) mm, rotated rx 180 ry 0 rz 0.01 deg; joints [33.055, -46.272, 104.847, -142.87, 64.681, 163.035]
  MoveL 2357 to (-215.4, 120.42, -12.92) mm, rotated rx 180 ry 0 rz 0.01 deg; joints [32.916, -46.016, 104.335, -142.944, 64.433, 162.929]
  MoveL 2358 to (-218, 114.35, -13.16) mm, rotated rx 180 ry 0 rz 0.01 deg; joints [32.666, -46.046, 104.437, -143.227, 64.411, 163.092]
  MoveL 2359 to (-213.48, 109.54, -13.4) mm, rotated rx 180 ry 0 rz 0.01 deg; joints [32.604, -46.312, 105.029, -143.385, 64.653, 163.337]
  MoveL 2360 to (-207.26, 111.75, -13.65) mm, rotated rx -180 ry 0 rz 0.01 deg; joints [32.806, -46.479, 105.401, -143.23, 64.88, 163.38]
  MoveL 2361 to (-206.79, 118.34, -13.89) mm, rotated rx 180 ry 0 rz 0.01 deg; joints [33.029, -46.332, 105.106, -142.954, 64.831, 163.18]
  MoveL 2362 to (-212.64, 121.4, -14.14) mm, rotated rx 180 ry 0 rz 0.01 deg; joints [33.006, -46.032, 104.497, -142.891, 64.577, 162.985]
  MoveL 2363 to (-217.8, 117.28, -14.38) mm, rotated rx 180 ry 0 rz 0.01 deg; joints [32.766, -45.924, 104.303, -143.119, 64.433, 163.039]
  MoveL 2364 to (-216.08, 110.9, -14.62) mm, rotated rx -180 ry 0 rz 0.01 deg; joints [32.595, -46.122, 104.755, -143.371, 64.583, 163.286]
  MoveL 2365 to (-209.55, 109.92, -14.87) mm, rotated rx 180 ry 0 rz 0.01 deg; joints [32.699, -46.373, 105.311, -143.347, 64.86, 163.439]
  MoveL 2366 to (-206.03, 115.51, -15.11) mm, rotated rx 180 ry 0 rz 0.01 deg; joints [32.954, -46.362, 105.304, -143.08, 64.942, 163.325]
  MoveL 2367 to (-209.75, 120.97, -15.36) mm, rotated rx 180 ry 0 rz 0.01 deg; joints [33.053, -46.087, 104.741, -142.895, 64.743, 163.089]
  MoveL 2368 to (-216.24, 119.76, -15.6) mm, rotated rx -180 ry 0 rz 0.01 deg; joints [32.879, -45.862, 104.296, -143.016, 64.513, 163.023]
  MoveL 2369 to (-217.73, 113.32, -15.85) mm, rotated rx 180 ry 0 rz 0.01 deg; joints [32.64, -45.942, 104.502, -143.302, 64.538, 163.217]
  MoveL 2370 to (-212.43, 109.38, -16.09) mm, rotated rx -180 ry 0 rz 0.01 deg; joints [32.622, -46.216, 105.11, -143.416, 64.802, 163.446]
  MoveL 2371 to (-206.69, 112.65, -16.33) mm, rotated rx 180 ry 0 rz 0.01 deg; joints [32.849, -46.34, 105.391, -143.222, 64.997, 163.447]
  MoveL 2372 to (-207.39, 119.22, -16.58) mm, rotated rx -180 ry 0 rz 0.01 deg; joints [33.047, -46.151, 105.007, -142.959, 64.903, 163.227]
  MoveL 2373 to (-213.69, 121.21, -16.82) mm, rotated rx -180 ry 0 rz 0.01 deg; joints [32.979, -45.86, 104.417, -142.946, 64.643, 163.059]
  MoveL 2374 to (-218.04, 116.24, -17.07) mm, rotated rx 180 ry 0 rz 0.01 deg; joints [32.728, -45.801, 104.328, -143.2, 64.54, 163.154]
  MoveL 2375 to (-215.22, 110.26, -17.31) mm, rotated rx -180 ry 0 rz 0.01 deg; joints [32.594, -46.029, 104.845, -143.424, 64.73, 163.408]
  MoveL 2376 to (-208.62, 110.45, -17.55) mm, rotated rx -180 ry 0 rz 0.01 deg; joints [32.737, -46.256, 105.348, -143.35, 64.996, 163.524]
  MoveL 2377 to (-206.15, 116.57, -17.8) mm, rotated rx -180 ry 0 rz 0.01 deg; joints [32.988, -46.194, 105.233, -143.072, 65.03, 163.375]
  MoveL 2378 to (-210.76, 121.29, -18.04) mm, rotated rx 180 ry 0 rz 0.01 deg; joints [33.044, -45.903, 104.637, -142.928, 64.804, 163.147]
  MoveL 2379 to (-216.94, 118.95, -18.29) mm, rotated rx 180 ry 0 rz 0.01 deg; joints [32.84, -45.716, 104.273, -143.092, 64.599, 163.123]
  MoveL 2380 to (-217.27, 112.36, -18.53) mm, rotated rx -180 ry 0 rz 0.01 deg; joints [32.62, -45.842, 104.577, -143.373, 64.672, 163.342]
  MoveL 2381 to (-211.36, 109.41, -18.77) mm, rotated rx 180 ry 0 rz 0.01 deg; joints [32.647, -46.115, 105.183, -143.438, 64.949, 163.549]
  MoveL 2382 to (-206.29, 113.64, -19.02) mm, rotated rx -180 ry 0 rz 0.01 deg; joints [32.891, -46.192, 105.364, -143.212, 65.107, 163.507]
  MoveL 2383 to (-208.14, 119.98, -19.26) mm, rotated rx -180 ry 0 rz 0.01 deg; joints [33.057, -45.966, 104.902, -142.971, 64.969, 163.275]
  MoveL 2384 to (-214.69, 120.83, -19.51) mm, rotated rx -180 ry 0 rz 0.01 deg; joints [32.947, -45.693, 104.35, -143.007, 64.712, 163.14]
  MoveL 2385 to (-218.09, 115.17, -19.75) mm, rotated rx 180 ry 0 rz 0.01 deg; joints [32.694, -45.684, 104.368, -143.28, 64.655, 163.274]
  MoveL 2386 to (-214.27, 109.78, -19.99) mm, rotated rx 180 ry 0 rz 0.01 deg; joints [32.6, -45.936, 104.934, -143.469, 64.878, 163.525]
  MoveL 2387 to (-207.8, 111.13, -20.24) mm, rotated rx -180 ry 0 rz 0.01 deg; joints [32.778, -46.13, 105.369, -143.348, 65.125, 163.602]
  MoveL 2388 to (-206.44, 117.59, -20.48) mm, rotated rx 180 ry 0 rz 0.01 deg; joints [33.016, -46.02, 105.15, -143.068, 65.111, 163.422]
  MoveL 2389 to (-211.82, 121.43, -20.73) mm, rotated rx -180 ry 0 rz 0.01 deg; joints [33.027, -45.722, 104.539, -142.969, 64.865, 163.21]
  MoveL 2390 to (-217.49, 118.04, -20.97) mm, rotated rx -180 ry 0 rz 0.01 deg; joints [32.8, -45.578, 104.267, -143.171, 64.692, 163.229]
  MoveL 2391 to (-216.66, 111.49, -21.21) mm, rotated rx -180 ry 0 rz 0.01 deg; joints [32.606, -45.746, 104.659, -143.438, 64.812, 163.466]
  MoveL 2392 to (-210.32, 109.63, -21.46) mm, rotated rx -180 ry 0 rz 0.01 deg; joints [32.677, -46.008, 105.244, -143.453, 65.092, 163.645]
  MoveL 2393 to (-206.07, 114.68, -21.7) mm, rotated rx 180 ry 0 rz 0.01 deg; joints [32.93, -46.036, 105.32, -143.201, 65.208, 163.563]
  MoveL 2394 to (-209.01, 120.6, -21.95) mm, rotated rx -180 ry 0 rz 0.01 deg; joints [33.06, -45.781, 104.795, -142.989, 65.032, 163.325]
  MoveL 2395 to (-215.61, 120.28, -22.19) mm, rotated rx 180 ry 0 rz 0.01 deg; joints [32.912, -45.533, 104.297, -143.074, 64.787, 163.227]
  MoveL 2396 to (-217.96, 114.11, -22.43) mm, rotated rx -180 ry 0 rz 0.01 deg; joints [32.665, -45.574, 104.422, -143.358, 64.777, 163.396]
  MoveL 2397 to (-213.25, 109.48, -22.68) mm, rotated rx -180 ry 0 rz 0.01 deg; joints [32.613, -45.84, 105.019, -143.505, 65.027, 163.637]
  MoveL 2398 to (-207.12, 111.95, -22.92) mm, rotated rx 180 ry 0 rz 0.01 deg; joints [32.82, -45.996, 105.371, -143.341, 65.248, 163.672]
  MoveL 2399 to (-206.92, 118.55, -23.17) mm, rotated rx 180 ry 0 rz 0.01 deg; joints [33.039, -45.841, 105.055, -143.068, 65.186, 163.468]
  MoveL 2400 to (-212.89, 121.38, -23.41) mm, rotated rx 180 ry 0 rz 0.01 deg; joints [33.005, -45.544, 104.449, -143.017, 64.928, 163.278]
  MoveL 2401 to (-217.87, 117.04, -23.65) mm, rotated rx -180 ry 0 rz 0.01 deg; joints [32.762, -45.448, 104.278, -143.251, 64.793, 163.34]
  MoveL 2402 to (-215.89, 110.74, -23.9) mm, rotated rx 180 ry 0 rz 0.01 deg; joints [32.599, -45.651, 104.746, -143.496, 64.955, 163.589]
  MoveL 2403 to (-209.33, 110.02, -24.14) mm, rotated rx -180 ry 0 rz 0.01 deg; joints [32.712, -45.895, 105.291, -143.46, 65.232, 163.735]
  MoveL 2404 to (-206.04, 115.75, -24.39) mm, rotated rx 180 ry 0 rz 0.01 deg; joints [32.967, -45.873, 105.259, -143.19, 65.301, 163.614]
  MoveL 2405 to (-209.97, 121.06, -24.63) mm, rotated rx 180 ry 0 rz 0.01 deg; joints [33.056, -45.595, 104.687, -143.015, 65.093, 163.379]
  MoveL 2406 to (-216.41, 119.58, -24.87) mm, rotated rx 180 ry 0 rz 0.01 deg; joints [32.874, -45.38, 104.259, -143.146, 64.867, 163.321]
  MoveL 2407 to (-217.64, 113.09, -25.12) mm, rotated rx 180 ry 0 rz 0.01 deg; joints [32.64, -45.47, 104.488, -143.432, 64.906, 163.519]
  MoveL 2408 to (-212.19, 109.37, -25.36) mm, rotated rx 180 ry 0 rz 0.01 deg; joints [32.632, -45.742, 105.097, -143.533, 65.175, 163.744]
  MoveL 2409 to (-206.59, 112.87, -25.61) mm, rotated rx -180 ry 0 rz 0.01 deg; joints [32.863, -45.854, 105.356, -143.331, 65.362, 163.737]
  MoveL 2410 to (-207.55, 119.4, -25.85) mm, rotated rx -180 ry 0 rz 0.01 deg; joints [33.054, -45.658, 104.953, -143.074, 65.255, 163.514]
  MoveL 2411 to (-213.93, 121.14, -26.1) mm, rotated rx 180 ry 0 rz 0.01 deg; joints [32.977, -45.372, 104.37, -143.072, 64.993, 163.352]
  MoveL 2412 to (-218.07, 115.99, -26.34) mm, rotated rx -180 ry 0 rz 0.01 deg; joints [32.725, -45.325, 104.304, -143.331, 64.901, 163.455]
  MoveL 2413 to (-215.01, 110.14, -26.58) mm, rotated rx -180 ry 0 rz 0.01 deg; joints [32.599, -45.557, 104.834, -143.546, 65.102, 163.708]
  MoveL 2414 to (-208.43, 110.59, -26.83) mm, rotated rx 180 ry 0 rz 0.01 deg; joints [32.751, -45.775, 105.323, -143.461, 65.365, 163.817]
  MoveL 2415 to (-206.2, 116.81, -27.07) mm, rotated rx -180 ry 0 rz 0.01 deg; joints [33, -45.702, 105.183, -143.183, 65.387, 163.662]
  MoveL 2416 to (-211, 121.34, -27.32) mm, rotated rx -180 ry 0 rz 0.01 deg; joints [33.045, -45.411, 104.582, -143.049, 65.153, 163.436]
  MoveL 2417 to (-217.08, 118.75, -27.56) mm, rotated rx 180 ry 0 rz 0.01 deg; joints [32.835, -45.235, 104.238, -143.222, 64.954, 163.42]
  MoveL 2418 to (-217.15, 112.15, -27.8) mm, rotated rx 180 ry 0 rz 0.01 deg; joints [32.621, -45.37, 104.563, -143.5, 65.041, 163.643]
  MoveL 2419 to (-211.12, 109.44, -28.05) mm, rotated rx 180 ry 0 rz 0.01 deg; joints [32.658, -45.638, 105.166, -143.553, 65.321, 163.845]
  MoveL 2420 to (-206.23, 113.88, -28.29) mm, rotated rx -180 ry 0 rz 0.01 deg; joints [32.905, -45.704, 105.323, -143.32, 65.469, 163.795]
  MoveL 2421 to (-208.33, 120.14, -28.54) mm, rotated rx -180 ry 0 rz 0.01 deg; joints [33.063, -45.472, 104.845, -143.086, 65.32, 163.562]
  MoveL 2422 to (-214.91, 120.72, -28.78) mm, rotated rx 180 ry 0 rz 0.01 deg; joints [32.944, -45.206, 104.303, -143.134, 65.063, 163.433]
  MoveL 2423 to (-218.08, 114.93, -29.02) mm, rotated rx 180 ry 0 rz 0.01 deg; joints [32.692, -45.209, 104.346, -143.41, 65.017, 163.574]
  MoveL 2424 to (-214.04, 109.7, -29.27) mm, rotated rx 180 ry 0 rz 0.01 deg; joints [32.607, -45.462, 104.921, -143.588, 65.25, 163.823]
  MoveL 2425 to (-207.63, 111.3, -29.51) mm, rotated rx 180 ry 0 rz 0.01 deg; joints [32.792, -45.646, 105.337, -143.457, 65.493, 163.892]
  MoveL 2426 to (-206.54, 117.82, -29.76) mm, rotated rx -180 ry 0 rz 0.01 deg; joints [33.027, -45.526, 105.095, -143.178, 65.466, 163.708]
  MoveL 2427 to (-212.06, 121.43, -30) mm, rotated rx -180 ry 0 rz 0.01 deg; joints [33.027, -45.23, 104.484, -143.09, 65.213, 163.499]
  MoveL 2428 to (-214.07, 121.43, -30) mm, rotated rx -180 ry 0 rz 0.01 deg; joints [32.985, -45.157, 104.327, -143.111, 65.134, 163.463]
  MoveC 2429 to (-216, 120.32, -30) mm, rotated rx -180 ry 0 rz 0.01 deg; joints [32.91, -45.112, 104.233, -143.177, 65.072, 163.465] to (-216, 118.1, -30) mm, rotated rx 180 ry 0 rz 0.01 deg; joints [32.838, -45.163, 104.345, -143.269, 65.099, 163.538]
  MoveL 2430 to (-214.84, 116.09, -30) mm, rotated rx 180 ry 0 rz 0.01 deg; joints [32.797, -45.251, 104.537, -143.341, 65.169, 163.624]
  MoveC 2431 to (-213.8, 115.05, -30) mm, rotated rx 180 ry 0 rz 0.01 deg; joints [32.785, -45.312, 104.67, -143.373, 65.223, 163.677] to (-212.38, 114.67, -30) mm, rotated rx 180 ry 0 rz 0.01 deg; joints [32.803, -45.373, 104.799, -143.374, 65.284, 163.714]
  MoveL 2432 to (-181.12, 114.67, -30) mm, rotated rx 180 ry 0 rz 0.01 deg; joints [33.466, -46.494, 107.197, -143.023, 66.504, 164.261]
  MoveC 2433 to (-179.7, 115.05, -30) mm, rotated rx 180 ry 0 rz 0.01 deg; joints [33.509, -46.536, 107.286, -142.99, 66.554, 164.274] to (-178.66, 116.08, -30) mm, rotated rx 180 ry 0 rz 0.01 deg; joints [33.565, -46.549, 107.312, -142.935, 66.581, 164.259]
  MoveL 2434 to (-177.5, 118.1, -30) mm, rotated rx -180 ry 0 rz 0.01 deg; joints [33.656, -46.545, 107.299, -142.838, 66.601, 164.214]
  MoveC 2435 to (-177.5, 120.32, -30) mm, rotated rx -180 ry 0 rz 0.01 deg; joints [33.729, -46.495, 107.188, -142.746, 66.573, 164.143] to (-179.42, 121.43, -30) mm, rotated rx 180 ry 0 rz 0.01 deg; joints [33.723, -46.402, 106.986, -142.724, 66.485, 164.074]
  MoveL 2436 to (-212.06, 121.43, -30) mm, rotated rx -180 ry 0 rz 0.01 deg; joints [33.027, -45.23, 104.484, -143.09, 65.213, 163.499]
  MoveC 2437 to (-215.51, 122.48, -30) mm, rotated rx -180 ry 0 rz 0.01 deg; joints [32.989, -45.081, 104.162, -143.083, 65.065, 163.403] to (-217.78, 125.28, -30) mm, rotated rx -180 ry 0 rz 0.01 deg; joints [33.032, -44.933, 103.844, -142.99, 64.941, 163.27]
  MoveC 2438 to (-219.95, 128.12, -30) mm, rotated rx -180 ry 0 rz 0.01 deg; joints [33.077, -44.788, 103.53, -142.895, 64.82, 163.136] to (-223.26, 129.45, -30) mm, rotated rx -180 ry 0 rz 0.01 deg; joints [33.051, -44.635, 103.202, -142.873, 64.672, 163.032]
  MoveC 2439 to (-226.46, 129.8, -30) mm, rotated rx -180 ry 0 rz 0.01 deg; joints [32.996, -44.509, 102.933, -142.889, 64.541, 162.961] to (-229.65, 130.15, -30) mm, rotated rx -180 ry 0 rz 0.01 deg; joints [32.941, -44.382, 102.663, -142.906, 64.409, 162.891]
  MoveC 2440 to (-231.45, 129.23, -30) mm, rotated rx -180 ry 0 rz 0.01 deg; joints [32.875, -44.337, 102.568, -142.961, 64.349, 162.889] to (-231.34, 127.21, -30) mm, rotated rx 180 ry 0 rz 0.01 deg; joints [32.813, -44.387, 102.679, -143.044, 64.378, 162.958]
  MoveC 2441 to (-228.59, 123.27, -30) mm, rotated rx 180 ry 0 rz 0.01 deg; joints [32.744, -44.581, 103.097, -143.181, 64.536, 163.14] to (-225.98, 119.23, -30) mm, rotated rx 180 ry 0 rz 0.01 deg; joints [32.668, -44.77, 103.506, -143.323, 64.689, 163.321]
  MoveC 2442 to (-223.49, 115.12, -30) mm, rotated rx -180 ry 0 rz 0.01 deg; joints [32.587, -44.955, 103.909, -143.469, 64.838, 163.501] to (-221.06, 110.97, -30) mm, rotated rx -180 ry 0 rz 0.01 deg; joints [32.503, -45.138, 104.307, -143.617, 64.985, 163.68]
  MoveC 2443 to (-217.95, 107.86, -30) mm, rotated rx 180 ry 0 rz 0.01 deg; joints [32.467, -45.322, 104.704, -143.714, 65.146, 163.836] to (-213.71, 106.73, -30) mm, rotated rx -180 ry 0 rz 0.01 deg; joints [32.518, -45.503, 105.091, -143.718, 65.328, 163.948]
  MoveL 2444 to (-179.8, 106.73, -30) mm, rotated rx -180 ry 0 rz 0.01 deg; joints [33.234, -46.718, 107.692, -143.335, 66.653, 164.537]
  MoveC 2445 to (-175.56, 107.86, -30) mm, rotated rx 180 ry 0 rz 0.01 deg; joints [33.363, -46.842, 107.956, -143.236, 66.803, 164.573] to (-172.44, 110.97, -30) mm, rotated rx -180 ry 0 rz 0.01 deg; joints [33.533, -46.882, 108.036, -143.07, 66.884, 164.528]
  MoveC 2446 to (-170.01, 115.11, -30) mm, rotated rx -180 ry 0 rz 0.01 deg; joints [33.722, -46.875, 108.012, -142.869, 66.925, 164.438] to (-167.53, 119.22, -30) mm, rotated rx 180 ry 0 rz 0.01 deg; joints [33.911, -46.869, 107.992, -142.669, 66.969, 164.35]
  MoveC 2447 to (-164.94, 123.27, -30) mm, rotated rx -180 ry 0 rz 0.01 deg; joints [34.1, -46.868, 107.982, -142.47, 67.018, 164.265] to (-162.2, 127.21, -30) mm, rotated rx 180 ry 0 rz 0.01 deg; joints [34.289, -46.874, 107.987, -142.274, 67.073, 164.186]
  MoveC 2448 to (-162.09, 129.22, -30) mm, rotated rx -180 ry 0 rz 0.01 deg; joints [34.357, -46.831, 107.892, -142.19, 67.052, 164.123] to (-163.89, 130.14, -30) mm, rotated rx 180 ry 0 rz 0.01 deg; joints [34.347, -46.748, 107.711, -142.175, 66.972, 164.063]
  MoveC 2449 to (-167.57, 129.75, -30) mm, rotated rx 180 ry 0 rz 0.01 deg; joints [34.253, -46.629, 107.457, -142.237, 66.837, 164.012] to (-171.24, 129.34, -30) mm, rotated rx 180 ry 0 rz 0.01 deg; joints [34.159, -46.51, 107.203, -142.3, 66.702, 163.961]
  MoveC 2450 to (-174.92, 129.02, -30) mm, rotated rx -180 ry 0 rz 0.01 deg; joints [34.067, -46.387, 106.942, -142.358, 66.564, 163.907] to (-178.62, 128.91, -30) mm, rotated rx 180 ry 0 rz 0.01 deg; joints [33.983, -46.26, 106.668, -142.406, 66.424, 163.846]
  MoveL 2451 to (-214.9, 128.91, -30) mm, rotated rx 180 ry 0 rz 0.01 deg; joints [33.208, -44.955, 103.884, -142.81, 65.01, 163.202]
  MoveC 2452 to (-218.6, 129.02, -30) mm, rotated rx 180 ry 0 rz 0.01 deg; joints [33.134, -44.817, 103.589, -142.844, 64.863, 163.131] to (-222.29, 129.34, -30) mm, rotated rx 180 ry 0 rz 0.01 deg; joints [33.067, -44.674, 103.284, -142.868, 64.712, 163.053]
  MoveL 2453 to (-223.26, 129.45, -30) mm, rotated rx -180 ry 0 rz 0.01 deg; joints [33.051, -44.635, 103.202, -142.873, 64.672, 163.032]
  MoveC 2454 to (-226.33, 130.76, -30) mm, rotated rx -180 ry 0 rz 0.01 deg; joints [33.029, -44.491, 102.894, -142.848, 64.534, 162.932] to (-228.17, 133.54, -30) mm, rotated rx 180 ry 0 rz 0.01 deg; joints [33.08, -44.358, 102.606, -142.751, 64.427, 162.805]
  MoveC 2455 to (-229.98, 136.34, -30) mm, rotated rx 180 ry 0 rz 0.01 deg; joints [33.131, -44.226, 102.319, -142.652, 64.321, 162.677] to (-232.99, 137.75, -30) mm, rotated rx 180 ry 0 rz 0.01 deg; joints [33.113, -44.081, 102.008, -142.622, 64.184, 162.574]
  MoveC 2456 to (-240.22, 138.96, -30) mm, rotated rx 180 ry 0 rz 0.01 deg; joints [33.003, -43.781, 101.371, -142.638, 63.879, 162.398] to (-247.44, 140.26, -30) mm, rotated rx -180 ry 0 rz 0.01 deg; joints [32.897, -43.478, 100.725, -142.648, 63.573, 162.217]
  MoveC 2457 to (-249.16, 139.46, -30) mm, rotated rx 180 ry 0 rz 0.01 deg; joints [32.837, -43.432, 100.628, -142.695, 63.513, 162.211] to (-248.98, 137.58, -30) mm, rotated rx -180 ry 0 rz 0.01 deg; joints [32.781, -43.483, 100.74, -142.772, 63.543, 162.279]
  MoveC 2458 to (-246.16, 134.35, -30) mm, rotated rx -180 ry 0 rz 0.01 deg; joints [32.737, -43.665, 101.133, -142.882, 63.696, 162.442] to (-243.31, 131.16, -30) mm, rotated rx 180 ry 0 rz 0.01 deg; joints [32.694, -43.848, 101.525, -142.99, 63.849, 162.604]
  MoveC 2459 to (-240.52, 127.92, -30) mm, rotated rx -180 ry 0 rz 0.01 deg; joints [32.648, -44.028, 101.914, -143.1, 64.001, 162.765] to (-237.88, 124.55, -30) mm, rotated rx 180 ry 0 rz 0.01 deg; joints [32.595, -44.205, 102.296, -143.216, 64.148, 162.927]
  MoveC 2460 to (-234.39, 119.53, -30) mm, rotated rx -180 ry 0 rz 0.01 deg; joints [32.505, -44.451, 102.827, -143.392, 64.349, 163.158] to (-231.28, 114.26, -30) mm, rotated rx -180 ry 0 rz 0.01 deg; joints [32.4, -44.686, 103.338, -143.581, 64.537, 163.389]
  MoveC 2461 to (-228.33, 108.91, -30) mm, rotated rx 180 ry 0 rz 0.01 deg; joints [32.288, -44.916, 103.837, -143.775, 64.72, 163.617] to (-225.32, 103.6, -30) mm, rotated rx 180 ry 0 rz 0.01 deg; joints [32.177, -45.147, 104.338, -143.967, 64.905, 163.844]
  MoveC 2462 to (-222.21, 100.49, -30) mm, rotated rx -180 ry 0 rz 0.01 deg; joints [32.14, -45.33, 104.735, -144.065, 65.066, 164] to (-217.97, 99.35, -30) mm, rotated rx -180 ry 0 rz 0.01 deg; joints [32.189, -45.511, 105.123, -144.068, 65.249, 164.111]
  MoveL 2463 to (-175.55, 99.35, -30) mm, rotated rx 180 ry 0 rz 0.01 deg; joints [33.082, -47.031, 108.376, -143.588, 66.908, 164.842]
  MoveC 2464 to (-171.3, 100.49, -30) mm, rotated rx 180 ry 0 rz 0.01 deg; joints [33.212, -47.154, 108.64, -143.488, 67.057, 164.878] to (-168.19, 103.6, -30) mm, rotated rx 180 ry 0 rz 0.01 deg; joints [33.383, -47.195, 108.72, -143.321, 67.138, 164.833]
  MoveC 2465 to (-167.11, 105.55, -30) mm, rotated rx -180 ry 0 rz 0.01 deg; joints [33.471, -47.189, 108.705, -143.227, 67.156, 164.79] to (-166.08, 107.52, -30) mm, rotated rx -180 ry 0 rz 0.01 deg; joints [33.558, -47.181, 108.684, -143.132, 67.17, 164.745]
  MoveC 2466 to (-165.06, 109.5, -30) mm, rotated rx -180 ry 0 rz 0.01 deg; joints [33.646, -47.173, 108.662, -143.038, 67.185, 164.7] to (-163.98, 111.45, -30) mm, rotated rx 180 ry 0 rz 0.01 deg; joints [33.734, -47.167, 108.647, -142.944, 67.202, 164.657]
  MoveC 2467 to (-159.67, 118.38, -30) mm, rotated rx 180 ry 0 rz 0.01 deg; joints [34.057, -47.162, 108.621, -142.604, 67.28, 164.511] to (-154.91, 125.01, -30) mm, rotated rx -180 ry 0 rz 0.01 deg; joints [34.38, -47.176, 108.64, -142.27, 67.377, 164.381]
  MoveC 2468 to (-149.83, 131.39, -30) mm, rotated rx 180 ry 0 rz 0.01 deg; joints [34.702, -47.206, 108.692, -141.942, 67.489, 164.265] to (-144.51, 137.59, -30) mm, rotated rx 180 ry 0 rz 0.01 deg; joints [35.024, -47.245, 108.765, -141.618, 67.611, 164.157]
  MoveC 2469 to (-144.31, 139.47, -30) mm, rotated rx 180 ry 0 rz 0.01 deg; joints [35.089, -47.209, 108.683, -141.538, 67.594, 164.1] to (-146.03, 140.27, -30) mm, rotated rx -180 ry 0 rz 0.01 deg; joints [35.076, -47.132, 108.516, -141.529, 67.52, 164.045]
  MoveC 2470 to (-149.98, 139.5, -30) mm, rotated rx -180 ry 0 rz 0.01 deg; joints [34.962, -47.014, 108.265, -141.613, 67.381, 164.001] to (-153.91, 138.66, -30) mm, rotated rx 180 ry 0 rz 0.01 deg; joints [34.846, -46.898, 108.017, -141.698, 67.244, 163.96]
  MoveC 2471 to (-157.85, 137.89, -30) mm, rotated rx 180 ry 0 rz 0.01 deg; joints [34.732, -46.779, 107.765, -141.781, 67.104, 163.917] to (-161.83, 137.29, -30) mm, rotated rx 180 ry 0 rz 0.01 deg; joints [34.624, -46.655, 107.499, -141.856, 66.961, 163.867]
  MoveC 2472 to (-170.21, 136.5, -30) mm, rotated rx -180 ry 0 rz 0.01 deg; joints [34.413, -46.381, 106.914, -141.993, 66.652, 163.747] to (-178.62, 136.2, -30) mm, rotated rx -180 ry 0 rz 0.01 deg; joints [34.218, -46.092, 106.296, -142.107, 66.333, 163.609]
  MoveL 2473 to (-214.9, 136.2, -30) mm, rotated rx 180 ry 0 rz 0.01 deg; joints [33.441, -44.786, 103.511, -142.509, 64.921, 162.959]
  MoveC 2474 to (-223.1, 136.52, -30) mm, rotated rx 180 ry 0 rz 0.01 deg; joints [33.279, -44.477, 102.852, -142.578, 64.592, 162.798] to (-231.26, 137.48, -30) mm, rotated rx 180 ry 0 rz 0.01 deg; joints [33.14, -44.152, 102.159, -142.617, 64.256, 162.615]
  MoveC 2475 to (-232.12, 137.62, -30) mm, rotated rx -180 ry 0 rz 0.01 deg; joints [33.127, -44.116, 102.084, -142.619, 64.22, 162.595] to (-232.99, 137.75, -30) mm, rotated rx 180 ry 0 rz 0.01 deg; joints [33.113, -44.081, 102.008, -142.622, 64.184, 162.574]
  MoveC 2476 to (-235.7, 139.06, -30) mm, rotated rx 180 ry 0 rz 0.01 deg; joints [33.099, -43.949, 101.726, -142.593, 64.059, 162.479] to (-237.25, 141.62, -30) mm, rotated rx 180 ry 0 rz 0.01 deg; joints [33.148, -43.83, 101.469, -142.501, 63.966, 162.363]
  MoveC 2477 to (-238.79, 144.2, -30) mm, rotated rx 180 ry 0 rz 0.01 deg; joints [33.197, -43.711, 101.213, -142.408, 63.873, 162.246] to (-241.46, 145.55, -30) mm, rotated rx 180 ry 0 rz 0.01 deg; joints [33.185, -43.578, 100.928, -142.375, 63.749, 162.149]
  MoveC 2478 to (-243.44, 145.95, -30) mm, rotated rx 180 ry 0 rz 0.01 deg; joints [33.156, -43.494, 100.75, -142.376, 63.665, 162.098] to (-245.41, 146.37, -30) mm, rotated rx -180 ry 0 rz 0.01 deg; joints [33.129, -43.41, 100.57, -142.376, 63.58, 162.046]
  MoveC 2479 to (-260.25, 150.34, -30) mm, rotated rx 180 ry 0 rz 0.01 deg; joints [32.952, -42.748, 99.162, -142.333, 62.93, 161.622] to (-274.68, 155.62, -30) mm, rotated rx -180 ry 0 rz 0.01 deg; joints [32.827, -42.06, 97.699, -142.22, 62.275, 161.15]
  MoveC 2480 to (-276.24, 155.09, -30) mm, rotated rx -180 ry 0 rz 0.01 deg; joints [32.78, -42.012, 97.599, -142.253, 62.217, 161.138] to (-275.91, 153.48, -30) mm, rotated rx -180 ry 0 rz 0.01 deg; joints [32.737, -42.064, 97.712, -142.318, 62.25, 161.201]
  MoveC 2481 to (-266.9, 146.13, -30) mm, rotated rx -180 ry 0 rz 0.01 deg; joints [32.689, -42.593, 98.841, -142.56, 62.71, 161.638] to (-258.46, 138.12, -30) mm, rotated rx -180 ry 0 rz 0.01 deg; joints [32.607, -43.108, 99.946, -142.829, 63.151, 162.08]
  MoveC 2482 to (-250.62, 129.54, -30) mm, rotated rx 180 ry 0 rz 0.01 deg; joints [32.495, -43.609, 101.022, -143.122, 63.574, 162.522] to (-243.35, 120.46, -30) mm, rotated rx 180 ry 0 rz 0.01 deg; joints [32.353, -44.094, 102.067, -143.436, 63.977, 162.963]
  MoveC 2483 to (-241.13, 117.36, -30) mm, rotated rx -180 ry 0 rz 0.01 deg; joints [32.299, -44.248, 102.4, -143.545, 64.104, 163.107] to (-239.04, 114.18, -30) mm, rotated rx 180 ry 0 rz 0.01 deg; joints [32.24, -44.399, 102.727, -143.658, 64.227, 163.251]
  MoveC 2484 to (-237.04, 110.94, -30) mm, rotated rx -180 ry 0 rz 0.01 deg; joints [32.176, -44.547, 103.048, -143.775, 64.347, 163.394] to (-235.1, 107.66, -30) mm, rotated rx 180 ry 0 rz 0.01 deg; joints [32.109, -44.693, 103.365, -143.893, 64.464, 163.537]
  MoveC 2485 to (-233.6, 104.95, -30) mm, rotated rx 180 ry 0 rz 0.01 deg; joints [32.052, -44.81, 103.618, -143.992, 64.557, 163.652] to (-232.19, 102.21, -30) mm, rotated rx 180 ry 0 rz 0.01 deg; joints [31.992, -44.924, 103.865, -144.092, 64.647, 163.767]
  MoveC 2486 to (-230.77, 99.46, -30) mm, rotated rx -180 ry 0 rz 0.01 deg; joints [31.932, -45.037, 104.112, -144.193, 64.737, 163.881] to (-229.27, 96.76, -30) mm, rotated rx -180 ry 0 rz 0.01 deg; joints [31.874, -45.153, 104.363, -144.291, 64.83, 163.995]
  MoveC 2487 to (-226.17, 93.65, -30) mm, rotated rx 180 ry 0 rz 0.01 deg; joints [31.836, -45.336, 104.759, -144.39, 64.991, 164.15] to (-221.92, 92.51, -30) mm, rotated rx 180 ry 0 rz 0.01 deg; joints [31.885, -45.517, 105.148, -144.394, 65.175, 164.261]
  MoveL 2488 to (-171.6, 92.51, -30) mm, rotated rx -180 ry 0 rz 0.01 deg; joints [32.94, -47.318, 109.007, -143.822, 67.145, 165.122]
  MoveC 2489 to (-167.35, 93.65, -30) mm, rotated rx -180 ry 0 rz 0.01 deg; joints [33.07, -47.442, 109.271, -143.721, 67.294, 165.158] to (-164.24, 96.76, -30) mm, rotated rx 180 ry 0 rz 0.01 deg; joints [33.242, -47.482, 109.352, -143.553, 67.375, 165.113]
  MoveC 2490 to (-162.68, 99.57, -30) mm, rotated rx 180 ry 0 rz 0.01 deg; joints [33.369, -47.475, 109.331, -143.417, 67.399, 165.052] to (-161.2, 102.42, -30) mm, rotated rx 180 ry 0 rz 0.01 deg; joints [33.496, -47.463, 109.301, -143.28, 67.42, 164.988]
  MoveC 2491 to (-159.72, 105.28, -30) mm, rotated rx 180 ry 0 rz 0.01 deg; joints [33.624, -47.452, 109.27, -143.143, 67.441, 164.923] to (-158.16, 108.08, -30) mm, rotated rx -180 ry 0 rz 0.01 deg; joints [33.751, -47.444, 109.247, -143.007, 67.465, 164.862]
  MoveC 2492 to (-149.79, 120.93, -30) mm, rotated rx -180 ry 0 rz 0.01 deg; joints [34.361, -47.444, 109.224, -142.369, 67.622, 164.598] to (-140.11, 132.82, -30) mm, rotated rx -180 ry 0 rz 0.01 deg; joints [34.969, -47.505, 109.333, -141.753, 67.836, 164.385]
  MoveC 2493 to (-129.3, 143.68, -30) mm, rotated rx -180 ry 0 rz 0.01 deg; joints [35.571, -47.621, 109.561, -141.16, 68.101, 164.221] to (-117.55, 153.52, -30) mm, rotated rx 180 ry 0 rz 0.01 deg; joints [36.165, -47.785, 109.897, -140.593, 68.409, 164.105]
  MoveC 2494 to (-117.23, 155.13, -30) mm, rotated rx 180 ry 0 rz 0.01 deg; joints [36.224, -47.758, 109.835, -140.523, 68.4, 164.059] to (-118.78, 155.65, -30) mm, rotated rx 180 ry 0 rz 0.01 deg; joints [36.204, -47.694, 109.696, -140.525, 68.336, 164.015]
  MoveC 2495 to (-129.42, 151.59, -30) mm, rotated rx -180 ry 0 rz 0.01 deg; joints [35.824, -47.432, 109.141, -140.841, 67.996, 163.964] to (-140.33, 148.33, -30) mm, rotated rx 180 ry 0 rz 0.01 deg; joints [35.467, -47.139, 108.516, -141.124, 67.632, 163.882]
  MoveC 2496 to (-151.44, 145.83, -30) mm, rotated rx -180 ry 0 rz 0.01 deg; joints [35.133, -46.816, 107.83, -141.374, 67.247, 163.771] to (-162.68, 144.04, -30) mm, rotated rx 180 ry 0 rz 0.01 deg; joints [34.823, -46.469, 107.088, -141.591, 66.844, 163.633]
  MoveC 2497 to (-170.63, 143.29, -30) mm, rotated rx 180 ry 0 rz 0.01 deg; joints [34.622, -46.208, 106.532, -141.72, 66.551, 163.518] to (-178.62, 143.05, -30) mm, rotated rx 180 ry 0 rz 0.01 deg; joints [34.438, -45.933, 105.943, -141.827, 66.248, 163.385]
  MoveL 2498 to (-214.9, 143.05, -30) mm, rotated rx 180 ry 0 rz 0.01 deg; joints [33.658, -44.626, 103.157, -142.226, 64.837, 162.73]
  MoveC 2499 to (-228.24, 143.67, -30) mm, rotated rx 180 ry 0 rz 0.01 deg; joints [33.398, -44.118, 102.077, -142.332, 64.301, 162.462] to (-241.46, 145.55, -30) mm, rotated rx -180 ry 0 rz 0.01 deg; joints [33.185, -43.578, 100.928, -142.375, 63.749, 162.149]
  MoveC 2500 to (-244.23, 147.01, -30) mm, rotated rx 180 ry 0 rz 0.01 deg; joints [33.174, -43.439, 100.63, -142.339, 63.62, 162.046] to (-245.72, 149.77, -30) mm, rotated rx -180 ry 0 rz 0.01 deg; joints [33.23, -43.317, 100.367, -142.237, 63.526, 161.923]
  MoveC 2501 to (-247.14, 152.55, -30) mm, rotated rx -180 ry 0 rz 0.01 deg; joints [33.287, -43.196, 100.106, -142.134, 63.435, 161.799] to (-249.82, 154.14, -30) mm, rotated rx -180 ry 0 rz 0.01 deg; joints [33.282, -43.056, 99.807, -142.09, 63.307, 161.692]
  MoveL 2502 to (-250.1, 154.21, -30) mm, rotated rx -180 ry 0 rz 0.01 deg; joints [33.278, -43.043, 99.78, -142.09, 63.295, 161.685]
  MoveC 2503 to (-267.01, 159.68, -30) mm, rotated rx -180 ry 0 rz 0.01 deg; joints [33.105, -42.26, 98.114, -141.995, 62.54, 161.16] to (-283.23, 166.95, -30) mm, rotated rx 180 ry 0 rz 0.01 deg; joints [33.005, -41.444, 96.382, -141.802, 61.784, 160.571]
  MoveC 2504 to (-285.49, 166.87, -30) mm, rotated rx -180 ry 0 rz 0.01 deg; joints [32.958, -41.356, 96.197, -141.82, 61.691, 160.527] to (-286.6, 164.9, -30) mm, rotated rx 180 ry 0 rz 0.01 deg; joints [32.876, -41.361, 96.211, -141.91, 61.669, 160.575]
  MoveL 2505 to (-286.6, 156.57, -30) mm, rotated rx 180 ry 0 rz 0.01 deg; joints [32.621, -41.567, 96.659, -142.261, 61.77, 160.875]
  MoveC 2506 to (-285.83, 153.43, -30) mm, rotated rx 180 ry 0 rz 0.01 deg; joints [32.54, -41.674, 96.89, -142.388, 61.839, 161.003] to (-283.71, 151, -30) mm, rotated rx 180 ry 0 rz 0.01 deg; joints [32.507, -41.818, 97.196, -142.476, 61.957, 161.133]
  MoveC 2507 to (-271.14, 141.15, -30) mm, rotated rx -180 ry 0 rz 0.01 deg; joints [32.449, -42.547, 98.753, -142.801, 62.595, 161.729] to (-259.67, 130.06, -30) mm, rotated rx -180 ry 0 rz 0.01 deg; joints [32.33, -43.252, 100.264, -143.176, 63.199, 162.333]
  MoveC 2508 to (-249.46, 117.78, -30) mm, rotated rx 180 ry 0 rz 0.01 deg; joints [32.145, -43.925, 101.713, -143.602, 63.763, 162.939] to (-240.71, 104.42, -30) mm, rotated rx -180 ry 0 rz 0.01 deg; joints [31.892, -44.556, 103.079, -144.081, 64.277, 163.541]
  MoveC 2509 to (-238.75, 100.89, -30) mm, rotated rx 180 ry 0 rz 0.01 deg; joints [31.817, -44.709, 103.41, -144.21, 64.399, 163.692] to (-236.9, 97.29, -30) mm, rotated rx -180 ry 0 rz 0.01 deg; joints [31.738, -44.858, 103.734, -144.343, 64.517, 163.843]
  MoveC 2510 to (-235.05, 93.7, -30) mm, rotated rx -180 ry 0 rz 0.01 deg; joints [31.658, -45.006, 104.056, -144.475, 64.635, 163.992] to (-233.08, 90.16, -30) mm, rotated rx -180 ry 0 rz 0.01 deg; joints [31.582, -45.156, 104.384, -144.604, 64.756, 164.14]
  MoveC 2511 to (-229.98, 87.05, -30) mm, rotated rx 180 ry 0 rz 0.01 deg; joints [31.543, -45.339, 104.779, -144.703, 64.918, 164.295] to (-225.73, 85.92, -30) mm, rotated rx 180 ry 0 rz 0.01 deg; joints [31.591, -45.52, 105.168, -144.708, 65.102, 164.405]
  MoveL 2512 to (-167.8, 85.92, -30) mm, rotated rx 180 ry 0 rz 0.01 deg; joints [32.802, -47.593, 109.612, -144.047, 67.373, 165.389]
  MoveC 2513 to (-163.55, 87.05, -30) mm, rotated rx 180 ry 0 rz 0.01 deg; joints [32.932, -47.716, 109.875, -143.946, 67.522, 165.425] to (-160.44, 90.16, -30) mm, rotated rx 180 ry 0 rz 0.01 deg; joints [33.104, -47.757, 109.956, -143.777, 67.602, 165.381]
  MoveC 2514 to (-158.41, 93.8, -30) mm, rotated rx -180 ry 0 rz 0.01 deg; joints [33.271, -47.748, 109.93, -143.6, 67.634, 165.302] to (-156.49, 97.5, -30) mm, rotated rx -180 ry 0 rz 0.01 deg; joints [33.436, -47.734, 109.892, -143.422, 67.661, 165.219]
  MoveC 2515 to (-154.58, 101.2, -30) mm, rotated rx 180 ry 0 rz 0.01 deg; joints [33.602, -47.719, 109.852, -143.244, 67.687, 165.137] to (-152.55, 104.84, -30) mm, rotated rx -180 ry 0 rz 0.01 deg; joints [33.768, -47.708, 109.823, -143.067, 67.719, 165.057]
  MoveC 2516 to (-143.85, 118.09, -30) mm, rotated rx 180 ry 0 rz 0.01 deg; joints [34.401, -47.712, 109.805, -142.406, 67.881, 164.788] to (-133.69, 130.26, -30) mm, rotated rx 180 ry 0 rz 0.01 deg; joints [35.032, -47.781, 109.932, -141.768, 68.108, 164.575]
  MoveC 2517 to (-122.28, 141.25, -30) mm, rotated rx 180 ry 0 rz 0.01 deg; joints [35.656, -47.913, 110.194, -141.159, 68.391, 164.419] to (-109.81, 151.02, -30) mm, rotated rx -180 ry 0 rz 0.01 deg; joints [36.267, -48.101, 110.582, -140.58, 68.725, 164.317]
  MoveC 2518 to (-107.68, 153.45, -30) mm, rotated rx 180 ry 0 rz 0.01 deg; joints [36.396, -48.114, 110.606, -140.45, 68.771, 164.275] to (-106.91, 156.59, -30) mm, rotated rx -180 ry 0 rz 0.01 deg; joints [36.516, -48.066, 110.495, -140.312, 68.759, 164.187]
  MoveL 2519 to (-106.91, 164.9, -30) mm, rotated rx 180 ry 0 rz 0.01 deg; joints [36.784, -47.869, 110.056, -139.977, 68.652, 163.918]
  MoveC 2520 to (-108.02, 166.87, -30) mm, rotated rx -180 ry 0 rz 0.01 deg; joints [36.82, -47.785, 109.873, -139.915, 68.587, 163.835] to (-110.28, 166.93, -30) mm, rotated rx 180 ry 0 rz 0.01 deg; joints [36.768, -47.709, 109.708, -139.946, 68.504, 163.794]
  MoveC 2521 to (-122.96, 161.03, -30) mm, rotated rx 180 ry 0 rz 0.01 deg; joints [36.279, -47.426, 109.111, -140.368, 68.114, 163.768] to (-136.16, 156.37, -30) mm, rotated rx -180 ry 0 rz 0.01 deg; joints [35.821, -47.091, 108.4, -140.741, 67.685, 163.692]
  MoveC 2522 to (-149.71, 152.91, -30) mm, rotated rx -180 ry 0 rz 0.01 deg; joints [35.4, -46.71, 107.588, -141.063, 67.223, 163.57] to (-163.5, 150.59, -30) mm, rotated rx -180 ry 0 rz 0.01 deg; joints [35.014, -46.286, 106.686, -141.334, 66.731, 163.404]
  MoveC 2523 to (-171.05, 149.88, -30) mm, rotated rx 180 ry 0 rz 0.01 deg; joints [34.823, -46.039, 106.159, -141.456, 66.453, 163.294] to (-178.62, 149.64, -30) mm, rotated rx 180 ry 0 rz 0.01 deg; joints [34.648, -45.778, 105.6, -141.557, 66.166, 163.167]
  MoveL 2524 to (-214.9, 149.64, -30) mm, rotated rx -180 ry 0 rz 0.01 deg; joints [33.866, -44.47, 102.814, -141.954, 64.756, 162.508]
  MoveC 2525 to (-232.5, 150.77, -30) mm, rotated rx 180 ry 0 rz 0.01 deg; joints [33.533, -43.79, 101.369, -142.078, 64.044, 162.14] to (-249.82, 154.14, -30) mm, rotated rx 180 ry 0 rz 0.01 deg; joints [33.282, -43.056, 99.807, -142.09, 63.307, 161.692]
  MoveC 2526 to (-253.02, 156.11, -30) mm, rotated rx -180 ry 0 rz 0.01 deg; joints [33.277, -42.886, 99.444, -142.035, 63.154, 161.562] to (-254.59, 159.52, -30) mm, rotated rx -180 ry 0 rz 0.01 deg; joints [33.351, -42.743, 99.135, -141.905, 63.049, 161.411]
  MoveC 2527 to (-256.09, 162.95, -30) mm, rotated rx 180 ry 0 rz 0.01 deg; joints [33.427, -42.602, 98.831, -141.775, 62.946, 161.261] to (-259.17, 165.06, -30) mm, rotated rx 180 ry 0 rz 0.01 deg; joints [33.429, -42.431, 98.467, -141.711, 62.795, 161.125]
  MoveC 2528 to (-269.02, 168.75, -30) mm, rotated rx -180 ry 0 rz 0.01 deg; joints [33.343, -41.958, 97.462, -141.63, 62.348, 160.796] to (-278.58, 173.13, -30) mm, rotated rx -180 ry 0 rz 0.01 deg; joints [33.285, -41.474, 96.433, -141.512, 61.901, 160.443]
  MoveC 2529 to (-281.91, 174.95, -30) mm, rotated rx -180 ry 0 rz 0.01 deg; joints [33.274, -41.296, 96.057, -141.458, 61.741, 160.308] to (-285.1, 176.98, -30) mm, rotated rx 180 ry 0 rz 0.01 deg; joints [33.272, -41.118, 95.678, -141.392, 61.584, 160.167]
  MoveC 2530 to (-288.24, 179.11, -30) mm, rotated rx 180 ry 0 rz 0.01 deg; joints [33.274, -40.939, 95.298, -141.322, 61.427, 160.023] to (-291.41, 181.19, -30) mm, rotated rx 180 ry 0 rz 0.01 deg; joints [33.274, -40.76, 94.917, -141.253, 61.27, 159.88]
  MoveC 2531 to (-293.58, 181.27, -30) mm, rotated rx 180 ry 0 rz 0.01 deg; joints [33.234, -40.67, 94.729, -141.262, 61.178, 159.83] to (-294.69, 179.41, -30) mm, rotated rx 180 ry 0 rz 0.01 deg; joints [33.156, -40.673, 94.738, -141.347, 61.155, 159.875]
  MoveL 2532 to (-294.69, 153.8, -30) mm, rotated rx 180 ry 0 rz 0.01 deg; joints [32.378, -41.313, 96.128, -142.428, 61.465, 160.809]
  MoveC 2533 to (-293.59, 149.35, -30) mm, rotated rx 180 ry 0 rz 0.01 deg; joints [32.263, -41.466, 96.457, -142.609, 61.565, 160.99] to (-290.55, 145.92, -30) mm, rotated rx 180 ry 0 rz 0.01 deg; joints [32.216, -41.67, 96.893, -142.734, 61.733, 161.174]
  MoveC 2534 to (-271.42, 130.25, -30) mm, rotated rx -180 ry 0 rz 0.01 deg; joints [32.103, -42.794, 99.295, -143.26, 62.715, 162.101] to (-255.11, 111.67, -30) mm, rotated rx 180 ry 0 rz 0.01 deg; joints [31.837, -43.85, 101.565, -143.907, 63.607, 163.039]
  MoveC 2535 to (-251.23, 106.15, -30) mm, rotated rx 180 ry 0 rz 0.01 deg; joints [31.737, -44.122, 102.153, -144.104, 63.831, 163.294] to (-247.69, 100.4, -30) mm, rotated rx 180 ry 0 rz 0.01 deg; joints [31.623, -44.384, 102.721, -144.313, 64.044, 163.547]
  MoveC 2536 to (-245.15, 95.85, -30) mm, rotated rx 180 ry 0 rz 0.01 deg; joints [31.526, -44.581, 103.148, -144.48, 64.201, 163.742] to (-242.72, 91.24, -30) mm, rotated rx 180 ry 0 rz 0.01 deg; joints [31.425, -44.774, 103.566, -144.65, 64.355, 163.935]
  MoveC 2537 to (-240.3, 86.63, -30) mm, rotated rx 180 ry 0 rz 0.01 deg; joints [31.322, -44.965, 103.983, -144.821, 64.508, 164.127] to (-237.75, 82.08, -30) mm, rotated rx -180 ry 0 rz 0.01 deg; joints [31.224, -45.159, 104.404, -144.987, 64.665, 164.317]
  MoveC 2538 to (-234.65, 78.97, -30) mm, rotated rx 180 ry 0 rz 0.01 deg; joints [31.184, -45.341, 104.799, -145.087, 64.828, 164.471] to (-230.41, 77.83, -30) mm, rotated rx -180 ry 0 rz 0.01 deg; joints [31.231, -45.523, 105.189, -145.093, 65.012, 164.581]
  MoveL 2539 to (-163.13, 77.83, -30) mm, rotated rx 180 ry 0 rz 0.01 deg; joints [32.631, -47.928, 110.349, -144.323, 67.652, 165.714]
  MoveC 2540 to (-158.88, 78.97, -30) mm, rotated rx 180 ry 0 rz 0.01 deg; joints [32.762, -48.051, 110.611, -144.22, 67.801, 165.749] to (-155.77, 82.08, -30) mm, rotated rx 180 ry 0 rz 0.01 deg; joints [32.934, -48.092, 110.693, -144.05, 67.881, 165.706]
  MoveC 2541 to (-153.16, 86.73, -30) mm, rotated rx 180 ry 0 rz 0.01 deg; joints [33.149, -48.082, 110.663, -143.823, 67.922, 165.607] to (-150.67, 91.44, -30) mm, rotated rx 180 ry 0 rz 0.01 deg; joints [33.362, -48.066, 110.619, -143.595, 67.958, 165.503]
  MoveC 2542 to (-148.18, 96.16, -30) mm, rotated rx 180 ry 0 rz 0.01 deg; joints [33.575, -48.048, 110.573, -143.367, 67.993, 165.399] to (-145.57, 100.81, -30) mm, rotated rx -180 ry 0 rz 0.01 deg; joints [33.789, -48.036, 110.537, -143.139, 68.034, 165.299]
  MoveC 2543 to (-136.97, 113.84, -30) mm, rotated rx 180 ry 0 rz 0.01 deg; joints [34.416, -48.041, 110.522, -142.486, 68.193, 165.037] to (-126.88, 125.75, -30) mm, rotated rx -180 ry 0 rz 0.01 deg; joints [35.041, -48.114, 110.656, -141.856, 68.418, 164.833]
  MoveC 2544 to (-115.51, 136.43, -30) mm, rotated rx 180 ry 0 rz 0.01 deg; joints [35.657, -48.25, 110.93, -141.255, 68.702, 164.686] to (-103.06, 145.85, -30) mm, rotated rx -180 ry 0 rz 0.01 deg; joints [36.26, -48.444, 111.332, -140.687, 69.037, 164.597]
  MoveC 2545 to (-99.95, 149.3, -30) mm, rotated rx 180 ry 0 rz 0.01 deg; joints [36.447, -48.466, 111.372, -140.5, 69.105, 164.539] to (-98.83, 153.81, -30) mm, rotated rx 180 ry 0 rz 0.01 deg; joints [36.62, -48.397, 111.215, -140.301, 69.088, 164.414]
  MoveL 2546 to (-98.83, 179.42, -30) mm, rotated rx -180 ry 0 rz 0.01 deg; joints [37.442, -47.786, 109.852, -139.273, 68.759, 163.582]
  MoveC 2547 to (-99.93, 181.28, -30) mm, rotated rx -180 ry 0 rz 0.01 deg; joints [37.474, -47.705, 109.673, -139.216, 68.695, 163.502] to (-102.1, 181.19, -30) mm, rotated rx -180 ry 0 rz 0.01 deg; joints [37.419, -47.636, 109.525, -139.252, 68.618, 163.467]
  MoveC 2548 to (-110.08, 176.28, -30) mm, rotated rx 180 ry 0 rz 0.01 deg; joints [37.071, -47.491, 109.222, -139.568, 68.391, 163.491] to (-118.3, 171.77, -30) mm, rotated rx -180 ry 0 rz 0.01 deg; joints [36.731, -47.326, 108.876, -139.868, 68.149, 163.497]
  MoveC 2549 to (-126.81, 167.8, -30) mm, rotated rx 180 ry 0 rz 0.01 deg; joints [36.404, -47.136, 108.475, -140.149, 67.887, 163.48] to (-135.6, 164.54, -30) mm, rotated rx 180 ry 0 rz 0.01 deg; joints [36.095, -46.916, 108.01, -140.403, 67.603, 163.434]
  MoveC 2550 to (-155.04, 159.78, -30) mm, rotated rx -180 ry 0 rz 0.01 deg; joints [35.498, -46.363, 106.832, -140.853, 66.936, 163.25] to (-174.98, 158, -30) mm, rotated rx 180 ry 0 rz 0.01 deg; joints [34.994, -45.708, 105.436, -141.172, 66.201, 162.954]
  MoveL 2551 to (-214.9, 157.73, -30) mm, rotated rx -180 ry 0 rz 0.01 deg; joints [34.12, -44.276, 102.388, -141.621, 64.657, 162.233]
  MoveC 2552 to (-231.39, 158.73, -30) mm, rotated rx 180 ry 0 rz 0.01 deg; joints [33.804, -43.641, 101.038, -141.738, 63.991, 161.888] to (-247.64, 161.71, -30) mm, rotated rx -180 ry 0 rz 0.01 deg; joints [33.561, -42.955, 99.58, -141.757, 63.303, 161.471]
  MoveC 2553 to (-253.44, 163.27, -30) mm, rotated rx 180 ry 0 rz 0.01 deg; joints [33.49, -42.695, 99.028, -141.74, 63.05, 161.302] to (-259.17, 165.06, -30) mm, rotated rx -180 ry 0 rz 0.01 deg; joints [33.429, -42.431, 98.467, -141.711, 62.795, 161.125]
  MoveC 2554 to (-262.2, 167.24, -30) mm, rotated rx 180 ry 0 rz 0.01 deg; joints [33.434, -42.26, 98.102, -141.643, 62.645, 160.988] to (-263.5, 170.73, -30) mm, rotated rx -180 ry 0 rz 0.01 deg; joints [33.515, -42.123, 97.807, -141.507, 62.549, 160.837]
  MoveC 2555 to (-264.72, 174.24, -30) mm, rotated rx 180 ry 0 rz 0.01 deg; joints [33.597, -41.989, 97.518, -141.37, 62.457, 160.687] to (-267.59, 176.58, -30) mm, rotated rx 180 ry 0 rz 0.01 deg; joints [33.61, -41.818, 97.154, -141.293, 62.311, 160.544]
  MoveC 2556 to (-271.37, 178.27, -30) mm, rotated rx 180 ry 0 rz 0.01 deg; joints [33.585, -41.628, 96.75, -141.249, 62.135, 160.406] to (-275.1, 180.07, -30) mm, rotated rx 180 ry 0 rz 0.01 deg; joints [33.565, -41.436, 96.342, -141.199, 61.96, 160.263]
  MoveC 2557 to (-281.53, 183.63, -30) mm, rotated rx -180 ry 0 rz 0.01 deg; joints [33.544, -41.091, 95.611, -141.091, 61.651, 159.998] to (-287.64, 187.72, -30) mm, rotated rx 180 ry 0 rz 0.01 deg; joints [33.545, -40.743, 94.871, -140.956, 61.347, 159.718]
  MoveC 2558 to (-293.53, 192.12, -30) mm, rotated rx -180 ry 0 rz 0.01 deg; joints [33.56, -40.393, 94.129, -140.804, 61.048, 159.428] to (-299.34, 196.62, -30) mm, rotated rx -180 ry 0 rz 0.01 deg; joints [33.579, -40.041, 93.381, -140.645, 60.749, 159.131]
  MoveC 2559 to (-301.41, 196.84, -30) mm, rotated rx 180 ry 0 rz 0.01 deg; joints [33.545, -39.951, 93.192, -140.646, 60.66, 159.077] to (-302.52, 195.08, -30) mm, rotated rx 180 ry 0 rz 0.01 deg; joints [33.471, -39.952, 93.197, -140.726, 60.635, 159.119]
  MoveL 2560 to (-302.51, 149.21, -30) mm, rotated rx -180 ry 0 rz 0.01 deg; joints [32.086, -41.111, 95.711, -142.667, 61.192, 160.812]
  MoveC 2561 to (-301.42, 144.94, -30) mm, rotated rx -180 ry 0 rz 0.01 deg; joints [31.976, -41.259, 96.029, -142.842, 61.289, 160.987] to (-298.4, 141.73, -30) mm, rotated rx 180 ry 0 rz 0.01 deg; joints [31.935, -41.458, 96.454, -142.96, 61.455, 161.164]
  MoveC 2562 to (-287.97, 134.37, -30) mm, rotated rx 180 ry 0 rz 0.01 deg; joints [31.909, -42.049, 97.713, -143.204, 61.98, 161.633] to (-278.31, 126.04, -30) mm, rotated rx 180 ry 0 rz 0.01 deg; joints [31.836, -42.625, 98.944, -143.487, 62.482, 162.112]
  MoveC 2563 to (-269.44, 116.86, -30) mm, rotated rx -180 ry 0 rz 0.01 deg; joints [31.72, -43.182, 100.139, -143.806, 62.958, 162.596] to (-261.38, 106.98, -30) mm, rotated rx 180 ry 0 rz 0.01 deg; joints [31.564, -43.717, 101.292, -144.156, 63.407, 163.079]
  MoveC 2564 to (-257.77, 101.84, -30) mm, rotated rx 180 ry 0 rz 0.01 deg; joints [31.47, -43.971, 101.839, -144.341, 63.616, 163.316] to (-254.47, 96.5, -30) mm, rotated rx 180 ry 0 rz 0.01 deg; joints [31.363, -44.215, 102.368, -144.536, 63.815, 163.552]
  MoveC 2565 to (-251.36, 90.97, -30) mm, rotated rx -180 ry 0 rz 0.01 deg; joints [31.245, -44.455, 102.888, -144.741, 64.007, 163.789] to (-248.37, 85.37, -30) mm, rotated rx 180 ry 0 rz 0.01 deg; joints [31.122, -44.69, 103.399, -144.948, 64.196, 164.024]
  MoveC 2566 to (-245.39, 79.78, -30) mm, rotated rx -180 ry 0 rz 0.01 deg; joints [30.998, -44.924, 103.907, -145.155, 64.384, 164.257] to (-242.28, 74.25, -30) mm, rotated rx -180 ry 0 rz 0.01 deg; joints [30.877, -45.159, 104.419, -145.358, 64.576, 164.488]
  MoveC 2567 to (-239.17, 71.14, -30) mm, rotated rx 180 ry 0 rz 0.01 deg; joints [30.836, -45.341, 104.813, -145.459, 64.739, 164.64] to (-234.93, 70, -30) mm, rotated rx 180 ry 0 rz 0.01 deg; joints [30.882, -45.523, 105.203, -145.466, 64.924, 164.75]
  MoveL 2568 to (-158.61, 70, -30) mm, rotated rx 180 ry 0 rz 0.01 deg; joints [32.463, -48.249, 111.057, -144.589, 67.922, 166.025]
  MoveC 2569 to (-154.36, 71.14, -30) mm, rotated rx 180 ry 0 rz 0.01 deg; joints [32.594, -48.371, 111.319, -144.486, 68.071, 166.06] to (-151.25, 74.25, -30) mm, rotated rx -180 ry 0 rz 0.01 deg; joints [32.768, -48.413, 111.402, -144.315, 68.151, 166.017]
  MoveL 2570 to (-138.79, 96.89, -30) mm, rotated rx -180 ry 0 rz 0.01 deg; joints [33.81, -48.352, 111.226, -143.207, 68.338, 165.532]
  MoveC 2571 to (-130.02, 110.03, -30) mm, rotated rx 180 ry 0 rz 0.01 deg; joints [34.448, -48.36, 111.217, -142.544, 68.501, 165.272] to (-119.63, 121.92, -30) mm, rotated rx -180 ry 0 rz 0.01 deg; joints [35.083, -48.442, 111.372, -141.907, 68.735, 165.074]
  MoveC 2572 to (-107.91, 132.49, -30) mm, rotated rx 180 ry 0 rz 0.01 deg; joints [35.707, -48.591, 111.675, -141.302, 69.031, 164.938] to (-95.11, 141.73, -30) mm, rotated rx 180 ry 0 rz 0.01 deg; joints [36.316, -48.8, 112.107, -140.73, 69.378, 164.86]
  MoveC 2573 to (-92.09, 144.97, -30) mm, rotated rx 180 ry 0 rz 0.01 deg; joints [36.495, -48.823, 112.152, -140.552, 69.446, 164.808] to (-91, 149.26, -30) mm, rotated rx -180 ry 0 rz 0.01 deg; joints [36.662, -48.759, 112.005, -140.362, 69.43, 164.69]
  MoveL 2574 to (-91, 195.08, -30) mm, rotated rx 180 ry 0 rz 0.01 deg; joints [38.127, -47.659, 109.549, -138.529, 68.839, 163.198]
  MoveC 2575 to (-92.1, 196.84, -30) mm, rotated rx 180 ry 0 rz 0.01 deg; joints [38.156, -47.579, 109.375, -138.476, 68.777, 163.12] to (-94.17, 196.62, -30) mm, rotated rx -180 ry 0 rz 0.01 deg; joints [38.098, -47.517, 109.242, -138.517, 68.705, 163.092]
  MoveC 2576 to (-104.35, 189.13, -30) mm, rotated rx 180 ry 0 rz 0.01 deg; joints [37.615, -47.367, 108.933, -138.969, 68.435, 163.165] to (-115.01, 182.36, -30) mm, rotated rx -180 ry 0 rz 0.01 deg; joints [37.145, -47.179, 108.542, -139.396, 68.134, 163.204]
  MoveC 2577 to (-126.24, 176.54, -30) mm, rotated rx 180 ry 0 rz 0.01 deg; joints [36.695, -46.944, 108.048, -139.789, 67.797, 163.201] to (-138.03, 171.98, -30) mm, rotated rx -180 ry 0 rz 0.01 deg; joints [36.275, -46.655, 107.436, -140.135, 67.418, 163.146]
  MoveC 2578 to (-156.88, 167.39, -30) mm, rotated rx -180 ry 0 rz 0.01 deg; joints [35.697, -46.117, 106.293, -140.567, 66.771, 162.964] to (-176.21, 165.73, -30) mm, rotated rx 180 ry 0 rz 0.01 deg; joints [35.211, -45.479, 104.934, -140.871, 66.058, 162.673]
  MoveL 2579 to (-214.9, 165.55, -30) mm, rotated rx 180 ry 0 rz 0.01 deg; joints [34.364, -44.087, 101.973, -141.299, 64.56, 161.965]
  MoveC 2580 to (-230.48, 166.49, -30) mm, rotated rx 180 ry 0 rz 0.01 deg; joints [34.064, -43.486, 100.695, -141.409, 63.932, 161.636] to (-245.85, 169.3, -30) mm, rotated rx -180 ry 0 rz 0.01 deg; joints [33.832, -42.837, 99.318, -141.427, 63.283, 161.239]
  MoveC 2581 to (-256.87, 172.49, -30) mm, rotated rx 180 ry 0 rz 0.01 deg; joints [33.704, -42.336, 98.253, -141.383, 62.798, 160.907] to (-267.59, 176.58, -30) mm, rotated rx 180 ry 0 rz 0.01 deg; joints [33.61, -41.818, 97.154, -141.293, 62.311, 160.544]
  MoveC 2582 to (-270.38, 178.95, -30) mm, rotated rx 180 ry 0 rz 0.01 deg; joints [33.626, -41.649, 96.794, -141.213, 62.167, 160.401] to (-271.34, 182.48, -30) mm, rotated rx 180 ry 0 rz 0.01 deg; joints [33.714, -41.522, 96.521, -141.072, 62.085, 160.253]
  MoveC 2583 to (-272.2, 186.01, -30) mm, rotated rx 180 ry 0 rz 0.01 deg; joints [33.803, -41.399, 96.255, -140.93, 62.006, 160.106] to (-274.79, 188.57, -30) mm, rotated rx -180 ry 0 rz 0.01 deg; joints [33.828, -41.232, 95.899, -140.841, 61.869, 159.959]
  MoveC 2584 to (-292.02, 200.08, -30) mm, rotated rx -180 ry 0 rz 0.01 deg; joints [33.827, -40.246, 93.808, -140.46, 61.013, 159.161] to (-307.1, 214.3, -30) mm, rotated rx 180 ry 0 rz 0.01 deg; joints [33.947, -39.254, 91.703, -139.931, 60.205, 158.28]
  MoveC 2585 to (-308.98, 214.76, -30) mm, rotated rx 180 ry 0 rz 0.01 deg; joints [33.924, -39.164, 91.513, -139.92, 60.12, 158.219] to (-310.08, 213.17, -30) mm, rotated rx -180 ry 0 rz 0.01 deg; joints [33.856, -39.161, 91.51, -139.992, 60.093, 158.256]
  MoveL 2586 to (-310.08, 144.56, -30) mm, rotated rx 180 ry 0 rz 0.01 deg; joints [31.799, -40.919, 95.313, -142.906, 60.928, 160.822]
  MoveC 2587 to (-308.98, 140.47, -30) mm, rotated rx -180 ry 0 rz 0.01 deg; joints [31.694, -41.062, 95.622, -143.074, 61.023, 160.991] to (-305.98, 137.48, -30) mm, rotated rx -180 ry 0 rz 0.01 deg; joints [31.659, -41.256, 96.034, -143.184, 61.186, 161.16]
  MoveC 2588 to (-295.01, 130.3, -30) mm, rotated rx 180 ry 0 rz 0.01 deg; joints [31.646, -41.866, 97.334, -143.422, 61.734, 161.635] to (-284.93, 121.92, -30) mm, rotated rx -180 ry 0 rz 0.01 deg; joints [31.579, -42.462, 98.606, -143.707, 62.256, 162.125]
  MoveC 2589 to (-275.74, 112.58, -30) mm, rotated rx -180 ry 0 rz 0.01 deg; joints [31.461, -43.036, 99.838, -144.034, 62.749, 162.621] to (-267.43, 102.45, -30) mm, rotated rx -180 ry 0 rz 0.01 deg; joints [31.3, -43.587, 101.024, -144.395, 63.213, 163.118]
  MoveC 2590 to (-264.08, 97.68, -30) mm, rotated rx 180 ry 0 rz 0.01 deg; joints [31.212, -43.823, 101.532, -144.568, 63.407, 163.338] to (-261.03, 92.72, -30) mm, rotated rx 180 ry 0 rz 0.01 deg; joints [31.112, -44.05, 102.023, -144.751, 63.592, 163.557]
  MoveL 2591 to (-246.65, 66.68, -30) mm, rotated rx -180 ry 0 rz 0.01 deg; joints [30.542, -45.156, 104.428, -145.717, 64.489, 164.651]
  MoveC 2592 to (-243.54, 63.58, -30) mm, rotated rx -180 ry 0 rz 0.01 deg; joints [30.5, -45.338, 104.821, -145.818, 64.652, 164.803] to (-239.3, 62.44, -30) mm, rotated rx 180 ry 0 rz 0.01 deg; joints [30.545, -45.52, 105.212, -145.826, 64.837, 164.912]
  MoveL 2593 to (-154.25, 62.44, -30) mm, rotated rx -180 ry 0 rz 0.01 deg; joints [32.299, -48.557, 111.737, -144.847, 68.183, 166.322]
  MoveC 2594 to (-150, 63.58, -30) mm, rotated rx 180 ry 0 rz 0.01 deg; joints [32.431, -48.679, 111.999, -144.742, 68.332, 166.357] to (-146.89, 66.68, -30) mm, rotated rx 180 ry 0 rz 0.01 deg; joints [32.605, -48.72, 112.082, -144.57, 68.411, 166.314]
  MoveL 2595 to (-132.24, 93.11, -30) mm, rotated rx 180 ry 0 rz 0.01 deg; joints [33.83, -48.655, 111.889, -143.271, 68.632, 165.755]
  MoveC 2596 to (-123.36, 106.32, -30) mm, rotated rx -180 ry 0 rz 0.01 deg; joints [34.477, -48.665, 111.884, -142.6, 68.796, 165.496] to (-112.78, 118.22, -30) mm, rotated rx 180 ry 0 rz 0.01 deg; joints [35.12, -48.753, 112.051, -141.956, 69.035, 165.303]
  MoveC 2597 to (-100.75, 128.65, -30) mm, rotated rx -180 ry 0 rz 0.01 deg; joints [35.75, -48.914, 112.381, -141.348, 69.342, 165.178] to (-87.52, 137.51, -30) mm, rotated rx -180 ry 0 rz 0.01 deg; joints [36.361, -49.143, 112.859, -140.781, 69.707, 165.119]
  MoveC 2598 to (-84.53, 140.53, -30) mm, rotated rx 180 ry 0 rz 0.01 deg; joints [36.533, -49.171, 112.913, -140.611, 69.776, 165.074] to (-83.43, 144.64, -30) mm, rotated rx -180 ry 0 rz 0.01 deg; joints [36.695, -49.111, 112.776, -140.427, 69.762, 164.963]
  MoveL 2599 to (-83.43, 213.16, -30) mm, rotated rx -180 ry 0 rz 0.01 deg; joints [38.878, -47.452, 109.073, -137.696, 68.876, 162.722]
  MoveC 2600 to (-84.54, 214.76, -30) mm, rotated rx -180 ry 0 rz 0.01 deg; joints [38.9, -47.376, 108.907, -137.65, 68.816, 162.649] to (-86.42, 214.3, -30) mm, rotated rx 180 ry 0 rz 0.01 deg; joints [38.839, -47.326, 108.802, -137.698, 68.755, 162.631]
  MoveC 2601 to (-103.22, 198.76, -30) mm, rotated rx -180 ry 0 rz 0.01 deg; joints [37.943, -47.166, 108.484, -138.568, 68.352, 162.862] to (-122.75, 186.81, -30) mm, rotated rx 180 ry 0 rz 0.01 deg; joints [37.101, -46.811, 107.744, -139.328, 67.794, 162.92]
  MoveC 2602 to (-144.07, 178.57, -30) mm, rotated rx 180 ry 0 rz 0.01 deg; joints [36.343, -46.288, 106.64, -139.95, 67.11, 162.819] to (-166.43, 173.88, -30) mm, rotated rx 180 ry 0 rz 0.01 deg; joints [35.685, -45.626, 105.234, -140.423, 66.328, 162.575]
  MoveL 2603 to (-214.9, 173.12, -30) mm, rotated rx 180 ry 0 rz 0.01 deg; joints [34.599, -43.902, 101.567, -140.988, 64.467, 161.703]
  MoveC 2604 to (-245.82, 177.04, -30) mm, rotated rx 180 ry 0 rz 0.01 deg; joints [34.07, -42.646, 98.9, -141.106, 63.189, 160.965] to (-274.79, 188.57, -30) mm, rotated rx 180 ry 0 rz 0.01 deg; joints [33.828, -41.232, 95.899, -140.841, 61.869, 159.959]
  MoveC 2605 to (-277.26, 191.11, -30) mm, rotated rx 180 ry 0 rz 0.01 deg; joints [33.855, -41.069, 95.552, -140.75, 61.736, 159.813] to (-277.89, 194.61, -30) mm, rotated rx -180 ry 0 rz 0.01 deg; joints [33.946, -40.954, 95.303, -140.608, 61.667, 159.67]
  MoveC 2606 to (-278.46, 198.09, -30) mm, rotated rx 180 ry 0 rz 0.01 deg; joints [34.039, -40.841, 95.06, -140.465, 61.601, 159.529] to (-280.79, 200.75, -30) mm, rotated rx -180 ry 0 rz 0.01 deg; joints [34.071, -40.679, 94.716, -140.368, 61.472, 159.38]
  MoveC 2607 to (-284.97, 203.56, -30) mm, rotated rx -180 ry 0 rz 0.01 deg; joints [34.071, -40.438, 94.206, -140.274, 61.264, 159.184] to (-289.05, 206.52, -30) mm, rotated rx -180 ry 0 rz 0.01 deg; joints [34.077, -40.197, 93.693, -140.173, 61.058, 158.983]
  MoveC 2608 to (-296.4, 212.79, -30) mm, rotated rx -180 ry 0 rz 0.01 deg; joints [34.115, -39.732, 92.708, -139.946, 60.674, 158.581] to (-302.97, 219.88, -30) mm, rotated rx 180 ry 0 rz 0.01 deg; joints [34.192, -39.273, 91.734, -139.677, 60.311, 158.158]
  MoveC 2609 to (-308.89, 227.5, -30) mm, rotated rx -180 ry 0 rz 0.01 deg; joints [34.297, -38.82, 90.774, -139.377, 59.967, 157.722] to (-314.38, 235.43, -30) mm, rotated rx -180 ry 0 rz 0.01 deg; joints [34.418, -38.372, 89.823, -139.058, 59.635, 157.277]
  MoveC 2610 to (-316.1, 236.07, -30) mm, rotated rx 180 ry 0 rz 0.01 deg; joints [34.402, -38.282, 89.634, -139.037, 59.554, 157.21] to (-317.19, 234.6, -30) mm, rotated rx 180 ry 0 rz 0.01 deg; joints [34.338, -38.277, 89.626, -139.103, 59.526, 157.243]
  MoveL 2611 to (-317.19, 140.21, -30) mm, rotated rx 180 ry 0 rz 0.01 deg; joints [31.531, -40.735, 94.933, -143.128, 60.677, 160.83]
  MoveC 2612 to (-316.06, 136.12, -30) mm, rotated rx -180 ry 0 rz 0.01 deg; joints [31.427, -40.88, 95.245, -143.296, 60.774, 161.001] to (-312.98, 133.2, -30) mm, rotated rx -180 ry 0 rz 0.01 deg; joints [31.395, -41.075, 95.661, -143.404, 60.941, 161.169]
  MoveC 2613 to (-292.25, 119.09, -30) mm, rotated rx -180 ry 0 rz 0.01 deg; joints [31.349, -42.239, 98.14, -143.877, 61.984, 162.08] to (-275.09, 100.8, -30) mm, rotated rx 180 ry 0 rz 0.01 deg; joints [31.099, -43.329, 100.479, -144.524, 62.916, 163.03]
  MoveC 2614 to (-273, 97.97, -30) mm, rotated rx -180 ry 0 rz 0.01 deg; joints [31.049, -43.473, 100.79, -144.627, 63.036, 163.163] to (-270.96, 95.1, -30) mm, rotated rx 180 ry 0 rz 0.01 deg; joints [30.996, -43.616, 101.098, -144.732, 63.155, 163.296]
  MoveC 2615 to (-269.01, 92.18, -30) mm, rotated rx 180 ry 0 rz 0.01 deg; joints [30.94, -43.756, 101.4, -144.839, 63.27, 163.429] to (-267.19, 89.17, -30) mm, rotated rx 180 ry 0 rz 0.01 deg; joints [30.878, -43.892, 101.696, -144.951, 63.381, 163.561]
  MoveL 2616 to (-250.74, 59.54, -30) mm, rotated rx 180 ry 0 rz 0.01 deg; joints [30.226, -45.153, 104.435, -146.055, 64.407, 164.806]
  MoveC 2617 to (-247.66, 56.45, -30) mm, rotated rx 180 ry 0 rz 0.01 deg; joints [30.183, -45.334, 104.825, -146.156, 64.569, 164.956] to (-243.45, 55.32, -30) mm, rotated rx -180 ry 0 rz 0.01 deg; joints [30.227, -45.514, 105.214, -146.164, 64.754, 165.063]
  MoveL 2618 to (-150.08, 55.32, -30) mm, rotated rx -180 ry 0 rz 0.01 deg; joints [32.145, -48.846, 112.378, -145.087, 68.431, 166.6]
  MoveC 2619 to (-145.88, 56.45, -30) mm, rotated rx 180 ry 0 rz 0.01 deg; joints [32.275, -48.966, 112.635, -144.983, 68.577, 166.634] to (-142.81, 59.52, -30) mm, rotated rx 180 ry 0 rz 0.01 deg; joints [32.448, -49.007, 112.718, -144.813, 68.656, 166.593]
  MoveL 2620 to (-126.09, 89.55, -30) mm, rotated rx 180 ry 0 rz 0.01 deg; joints [33.849, -48.939, 112.51, -143.33, 68.907, 165.964]
  MoveC 2621 to (-106.38, 114.67, -30) mm, rotated rx -180 ry 0 rz 0.01 deg; joints [35.151, -49.043, 112.687, -142.005, 69.316, 165.519] to (-80.45, 133.3, -30) mm, rotated rx -180 ry 0 rz 0.01 deg; joints [36.394, -49.467, 113.57, -140.837, 70.016, 165.368]
  MoveC 2622 to (-77.43, 136.14, -30) mm, rotated rx 180 ry 0 rz 0.01 deg; joints [36.562, -49.499, 113.634, -140.672, 70.087, 165.329] to (-76.32, 140.14, -30) mm, rotated rx -180 ry 0 rz 0.01 deg; joints [36.721, -49.443, 113.505, -140.492, 70.075, 165.222]
  MoveL 2623 to (-76.32, 234.6, -30) mm, rotated rx 180 ry 0 rz 0.01 deg; joints [39.714, -47.132, 108.35, -136.743, 68.851, 162.114]
  MoveC 2624 to (-77.42, 236.07, -30) mm, rotated rx 180 ry 0 rz 0.01 deg; joints [39.731, -47.059, 108.19, -136.703, 68.794, 162.044] to (-79.14, 235.43, -30) mm, rotated rx -180 ry 0 rz 0.01 deg; joints [39.668, -47.02, 108.108, -136.755, 68.741, 162.035]
  MoveC 2625 to (-85.59, 226.33, -30) mm, rotated rx -180 ry 0 rz 0.01 deg; joints [39.229, -47.046, 108.179, -137.211, 68.63, 162.235] to (-92.79, 217.81, -30) mm, rotated rx 180 ry 0 rz 0.01 deg; joints [38.789, -47.029, 108.158, -137.657, 68.483, 162.4]
  MoveC 2626 to (-100.72, 209.96, -30) mm, rotated rx 180 ry 0 rz 0.01 deg; joints [38.352, -46.968, 108.04, -138.087, 68.299, 162.527] to (-109.35, 202.88, -30) mm, rotated rx 180 ry 0 rz 0.01 deg; joints [37.923, -46.86, 107.82, -138.494, 68.078, 162.615]
  MoveC 2627 to (-120.71, 195.51, -30) mm, rotated rx 180 ry 0 rz 0.01 deg; joints [37.421, -46.664, 107.414, -138.951, 67.758, 162.663] to (-132.91, 189.65, -30) mm, rotated rx -180 ry 0 rz 0.01 deg; joints [36.95, -46.397, 106.853, -139.355, 67.384, 162.644]
  MoveC 2628 to (-145.69, 185.23, -30) mm, rotated rx 180 ry 0 rz 0.01 deg; joints [36.514, -46.069, 106.159, -139.703, 66.966, 162.565] to (-158.86, 182.14, -30) mm, rotated rx -180 ry 0 rz 0.01 deg; joints [36.115, -45.689, 105.353, -139.995, 66.511, 162.433]
  MoveC 2629 to (-172.79, 180.33, -30) mm, rotated rx -180 ry 0 rz 0.01 deg; joints [35.744, -45.244, 104.408, -140.237, 66.006, 162.24] to (-186.84, 179.93, -30) mm, rotated rx 180 ry 0 rz 0.01 deg; joints [35.419, -44.754, 103.366, -140.414, 65.474, 161.995]
  MoveL 2630 to (-214.9, 180.23, -30) mm, rotated rx -180 ry 0 rz 0.01 deg; joints [34.819, -43.726, 101.182, -140.695, 64.379, 161.456]
  MoveC 2631 to (-234.82, 182.02, -30) mm, rotated rx -180 ry 0 rz 0.01 deg; joints [34.451, -42.938, 99.51, -140.806, 63.568, 161.006] to (-254.11, 187.33, -30) mm, rotated rx 180 ry 0 rz 0.01 deg; joints [34.212, -42.069, 97.666, -140.745, 62.728, 160.43]
  MoveC 2632 to (-267.81, 193.32, -30) mm, rotated rx -180 ry 0 rz 0.01 deg; joints [34.112, -41.384, 96.211, -140.595, 62.097, 159.93] to (-280.79, 200.75, -30) mm, rotated rx 180 ry 0 rz 0.01 deg; joints [34.071, -40.679, 94.716, -140.368, 61.472, 159.38]
  MoveC 2633 to (-282.75, 203.1, -30) mm, rotated rx 180 ry 0 rz 0.01 deg; joints [34.102, -40.539, 94.418, -140.281, 61.362, 159.249] to (-283.02, 206.15, -30) mm, rotated rx -180 ry 0 rz 0.01 deg; joints [34.187, -40.448, 94.222, -140.154, 61.313, 159.128]
  MoveC 2634 to (-283.2, 209.19, -30) mm, rotated rx -180 ry 0 rz 0.01 deg; joints [34.273, -40.361, 94.033, -140.028, 61.268, 159.01] to (-284.95, 211.67, -30) mm, rotated rx 180 ry 0 rz 0.01 deg; joints [34.312, -40.225, 93.743, -139.933, 61.165, 158.877]
  MoveC 2635 to (-304.57, 232.27, -30) mm, rotated rx 180 ry 0 rz 0.01 deg; joints [34.521, -38.867, 90.866, -139.157, 60.09, 157.634] to (-318.32, 257.17, -30) mm, rotated rx -180 ry 0 rz 0.01 deg; joints [34.961, -37.588, 88.153, -138.138, 59.196, 156.298]
  MoveC 2636 to (-321.49, 258.92, -30) mm, rotated rx 180 ry 0 rz 0.01 deg; joints [34.947, -37.403, 87.764, -138.07, 59.039, 156.146] to (-323.8, 256.13, -30) mm, rotated rx 180 ry 0 rz 0.01 deg; joints [34.823, -37.385, 87.731, -138.196, 58.975, 156.204]
  MoveL 2637 to (-323.79, 135.95, -30) mm, rotated rx -180 ry 0 rz 0.01 deg; joints [31.277, -40.567, 94.588, -143.341, 60.446, 160.845]
  MoveC 2638 to (-322.7, 132.06, -30) mm, rotated rx -180 ry 0 rz 0.01 deg; joints [31.178, -40.706, 94.886, -143.502, 60.539, 161.008] to (-319.74, 129.31, -30) mm, rotated rx -180 ry 0 rz 0.01 deg; joints [31.148, -40.893, 95.284, -143.604, 60.699, 161.168]
  MoveC 2639 to (-312.69, 125.47, -30) mm, rotated rx 180 ry 0 rz 0.01 deg; joints [31.161, -41.271, 96.087, -143.731, 61.045, 161.449] to (-305.84, 121.27, -30) mm, rotated rx 180 ry 0 rz 0.01 deg; joints [31.159, -41.646, 96.886, -143.87, 61.386, 161.735]
  MoveC 2640 to (-299.29, 116.61, -30) mm, rotated rx -180 ry 0 rz 0.01 deg; joints [31.137, -42.017, 97.676, -144.027, 61.718, 162.027] to (-293.17, 111.39, -30) mm, rotated rx -180 ry 0 rz 0.01 deg; joints [31.089, -42.38, 98.453, -144.208, 62.037, 162.327]
  MoveC 2641 to (-281.2, 98.29, -30) mm, rotated rx 180 ry 0 rz 0.01 deg; joints [30.902, -43.148, 100.1, -144.676, 62.693, 163] to (-271.42, 83.47, -30) mm, rotated rx 180 ry 0 rz 0.01 deg; joints [30.612, -43.855, 101.626, -145.225, 63.274, 163.671]
  MoveL 2642 to (-254.48, 52.79, -30) mm, rotated rx 180 ry 0 rz 0.01 deg; joints [29.93, -45.154, 104.448, -146.373, 64.333, 164.953]
  MoveC 2643 to (-251.6, 49.81, -30) mm, rotated rx -180 ry 0 rz 0.01 deg; joints [29.886, -45.324, 104.817, -146.472, 64.486, 165.096] to (-247.6, 48.72, -30) mm, rotated rx 180 ry 0 rz 0.01 deg; joints [29.927, -45.496, 105.187, -146.481, 64.662, 165.198]
  MoveL 2644 to (-145.89, 48.72, -30) mm, rotated rx -180 ry 0 rz 0.01 deg; joints [32.007, -49.123, 112.992, -145.306, 68.673, 166.861]
  MoveC 2645 to (-141.91, 49.81, -30) mm, rotated rx 180 ry 0 rz 0.01 deg; joints [32.132, -49.236, 113.235, -145.205, 68.811, 166.892] to (-139.05, 52.78, -30) mm, rotated rx 180 ry 0 rz 0.01 deg; joints [32.298, -49.273, 113.308, -145.041, 68.883, 166.851]
  MoveL 2646 to (-119.94, 86.45, -30) mm, rotated rx -180 ry 0 rz 0.01 deg; joints [33.884, -49.21, 113.104, -143.367, 69.176, 166.157]
  MoveC 2647 to (-108.72, 102.31, -30) mm, rotated rx 180 ry 0 rz 0.01 deg; joints [34.681, -49.239, 113.135, -142.546, 69.388, 165.859] to (-95.06, 116.12, -30) mm, rotated rx -180 ry 0 rz 0.01 deg; joints [35.468, -49.382, 113.417, -141.77, 69.711, 165.66]
  MoveC 2648 to (-90.12, 119.96, -30) mm, rotated rx 180 ry 0 rz 0.01 deg; joints [35.715, -49.456, 113.572, -141.534, 69.84, 165.622] to (-84.83, 123.33, -30) mm, rotated rx 180 ry 0 rz 0.01 deg; joints [35.955, -49.552, 113.773, -141.312, 69.988, 165.605]
  MoveC 2649 to (-79.37, 126.37, -30) mm, rotated rx 180 ry 0 rz 0.01 deg; joints [36.19, -49.659, 114, -141.1, 70.145, 165.601] to (-73.82, 129.27, -30) mm, rotated rx -180 ry 0 rz 0.01 deg; joints [36.422, -49.771, 114.237, -140.89, 70.306, 165.602]
  MoveC 2650 to (-70.83, 132.04, -30) mm, rotated rx 180 ry 0 rz 0.01 deg; joints [36.588, -49.804, 114.303, -140.728, 70.377, 165.565] to (-69.72, 135.96, -30) mm, rotated rx -180 ry 0 rz 0.01 deg; joints [36.746, -49.75, 114.178, -140.551, 70.365, 165.461]
  MoveL 2651 to (-69.72, 256.11, -30) mm, rotated rx 180 ry 0 rz 0.01 deg; joints [40.529, -46.778, 107.556, -135.801, 68.806, 161.481]
  MoveC 2652 to (-72.03, 258.9, -30) mm, rotated rx 180 ry 0 rz 0.01 deg; joints [40.554, -46.629, 107.233, -135.729, 68.69, 161.341] to (-75.2, 257.16, -30) mm, rotated rx 180 ry 0 rz 0.01 deg; joints [40.421, -46.574, 107.117, -135.847, 68.601, 161.346]
  MoveC 2653 to (-89, 232.32, -30) mm, rotated rx 180 ry 0 rz 0.01 deg; joints [39.327, -46.78, 107.599, -137.028, 68.432, 161.968] to (-108.73, 211.89, -30) mm, rotated rx -180 ry 0 rz 0.01 deg; joints [38.217, -46.653, 107.363, -138.128, 67.985, 162.319]
  MoveC 2654 to (-132.95, 197.08, -30) mm, rotated rx -180 ry 0 rz 0.01 deg; joints [37.18, -46.211, 106.443, -139.057, 67.289, 162.392] to (-160.04, 188.63, -30) mm, rotated rx 180 ry 0 rz 0.01 deg; joints [36.29, -45.487, 104.912, -139.747, 66.385, 162.19]
  MoveC 2655 to (-173.68, 186.87, -30) mm, rotated rx 180 ry 0 rz 0.01 deg; joints [35.927, -45.051, 103.986, -139.982, 65.89, 162] to (-187.43, 186.5, -30) mm, rotated rx 180 ry 0 rz 0.01 deg; joints [35.61, -44.57, 102.963, -140.153, 65.369, 161.757]
  MoveL 2656 to (-214.9, 186.83, -30) mm, rotated rx 180 ry 0 rz 0.01 deg; joints [35.021, -43.562, 100.822, -140.424, 64.298, 161.224]
  MoveC 2657 to (-252.06, 193.23, -30) mm, rotated rx 180 ry 0 rz 0.01 deg; joints [34.432, -41.998, 97.506, -140.484, 62.739, 160.258] to (-284.95, 211.67, -30) mm, rotated rx 180 ry 0 rz 0.01 deg; joints [34.312, -40.225, 93.743, -139.933, 61.165, 158.877]
